LIN {X 0.238,Y -427.107,Z 1023.933,A 0.000,B 0.000,C 90.000,E1 203.823} C_DIS
LIN {X -0.247,Y -422.074,Z 1023.919,A 0.000,B 0.000,C 90.000,E1 201.535} C_DIS
LIN {X 0.239,Y -416.335,Z 1023.903,A 0.000,B 0.000,C 90.000,E1 198.417} C_DIS
LIN {X -0.105,Y -409.408,Z 1023.878,A 0.000,B 0.000,C 90.000,E1 194.008} C_DIS
LIN {X -0.209,Y -406.791,Z 1023.866,A 0.000,B 0.000,C 90.000,E1 191.951} C_DIS
LIN {X -0.089,Y -405.984,Z 1023.860,A 0.000,B 0.000,C 90.000,E1 190.894} C_DIS
LIN {X -0.067,Y -405.858,Z 1023.857,A 0.000,B 0.000,C 90.000,E1 190.197} C_DIS
LIN {X 0.174,Y -406.074,Z 1023.856,A 0.000,B 0.000,C 90.000,E1 189.962} C_DIS
LIN {X 0.195,Y -406.543,Z 1023.852,A 0.000,B 0.000,C 90.000,E1 189.265} C_DIS
LIN {X 0.208,Y -407.205,Z 1023.850,A 0.000,B 0.000,C 90.000,E1 188.916} C_DIS
LIN {X -0.175,Y -408.954,Z 1023.847,A 0.000,B 0.000,C 90.000,E1 188.398} C_DIS
LIN {X -0.116,Y -411.971,Z 1023.843,A 0.000,B 0.000,C 90.000,E1 187.701} C_DIS
LIN {X -0.050,Y -416.031,Z 1023.839,A 0.000,B 0.000,C 90.000,E1 187.004} C_DIS
LIN {X 0.026,Y -419.441,Z 1023.836,A 0.000,B 0.000,C 90.000,E1 186.486} C_DIS
LIN {X -0.081,Y -428.211,Z 1023.830,A 0.000,B 0.000,C 90.000,E1 185.334} C_DIS
LIN {X -0.106,Y -440.088,Z 1023.821,A 0.000,B 0.000,C 90.000,E1 183.841} C_DIS
LIN {X -0.100,Y -449.299,Z 1023.815,A 0.000,B 0.000,C 90.000,E1 182.694} C_DIS
LIN {X -0.039,Y -460.677,Z 1023.807,A 0.000,B 0.000,C 90.000,E1 181.260} C_DIS
LIN {X 0.183,Y -467.926,Z 1023.802,A 0.000,B 0.000,C 90.000,E1 180.286} C_DIS
LIN {X 0.049,Y -474.878,Z 1023.797,A 0.000,B 0.000,C 90.000,E1 179.370} C_DIS
LIN {X 0.054,Y -482.712,Z 1023.791,A 0.000,B 0.000,C 90.000,E1 178.282} C_DIS
LIN {X -0.145,Y -488.160,Z 1023.786,A 0.000,B 0.000,C 90.000,E1 177.535} C_DIS
LIN {X -0.121,Y -494.546,Z 1023.781,A 0.000,B 0.000,C 90.000,E1 176.617} C_DIS
LIN {X -0.011,Y -502.317,Z 1023.775,A 0.000,B 0.000,C 90.000,E1 175.412} C_DIS
LIN {X 0.217,Y -508.156,Z 1023.770,A 0.000,B 0.000,C 90.000,E1 174.489} C_DIS
LIN {X -0.082,Y -515.532,Z 1023.763,A 0.000,B 0.000,C 90.000,E1 173.337} C_DIS
LIN {X -0.238,Y -525.703,Z 1023.753,A 0.000,B 0.000,C 90.000,E1 171.602} C_DIS
LIN {X -0.062,Y -533.859,Z 1023.745,A 0.000,B 0.000,C 90.000,E1 170.151} C_DIS
LIN {X -0.114,Y -541.353,Z 1023.738,A 0.000,B 0.000,C 90.000,E1 168.870} C_DIS
LIN {X -0.051,Y -548.610,Z 1023.731,A 0.000,B 0.000,C 90.000,E1 167.589} C_DIS
LIN {X 0.120,Y -554.019,Z 1023.726,A 0.000,B 0.000,C 90.000,E1 166.589} C_DIS
LIN {X -0.172,Y -561.522,Z 1023.718,A 0.000,B 0.000,C 90.000,E1 165.227} C_DIS
LIN {X -0.068,Y -568.191,Z 1023.711,A 0.000,B 0.000,C 90.000,E1 163.976} C_DIS
LIN {X 0.141,Y -574.462,Z 1023.704,A 0.000,B 0.000,C 90.000,E1 162.725} C_DIS
LIN {X -0.217,Y -578.394,Z 1023.700,A 0.000,B 0.000,C 90.000,E1 161.945} C_DIS
LIN {X 0.119,Y -582.822,Z 1023.694,A 0.000,B 0.000,C 90.000,E1 160.967} C_DIS
LIN {X -0.235,Y -586.875,Z 1023.689,A 0.000,B 0.000,C 90.000,E1 160.061} C_DIS
LIN {X 0.148,Y -591.422,Z 1023.683,A 0.000,B 0.000,C 90.000,E1 158.954} C_DIS
LIN {X -0.174,Y -595.674,Z 1023.677,A 0.000,B 0.000,C 90.000,E1 157.922} C_DIS
LIN {X 0.096,Y -598.641,Z 1023.673,A 0.000,B 0.000,C 90.000,E1 157.102} C_DIS
LIN {X 0.090,Y -602.279,Z 1023.667,A 0.000,B 0.000,C 90.000,E1 156.049} C_DIS
LIN {X -0.170,Y -605.727,Z 1023.661,A 0.000,B 0.000,C 90.000,E1 155.025} C_DIS
LIN {X -0.141,Y -609.702,Z 1023.654,A 0.000,B 0.000,C 90.000,E1 153.717} C_DIS
LIN {X -0.056,Y -613.370,Z 1023.647,A 0.000,B 0.000,C 90.000,E1 152.410} C_DIS
LIN {X -0.166,Y -616.159,Z 1023.641,A 0.000,B 0.000,C 90.000,E1 151.385} C_DIS
LIN {X 0.316,Y -620.763,Z 1023.631,A 0.000,B 0.000,C 90.000,E1 149.537} C_DIS
LIN {X -0.163,Y -626.030,Z 1023.620,A 0.000,B 0.000,C 90.000,E1 147.533} C_DIS
LIN {X 0.163,Y -630.398,Z 1023.610,A 0.000,B 0.000,C 90.000,E1 145.722} C_DIS
LIN {X 0.232,Y -634.076,Z 1023.601,A 0.000,B 0.000,C 90.000,E1 144.196} C_DIS
LIN {X -0.032,Y -636.564,Z 1023.596,A 0.000,B 0.000,C 90.000,E1 143.210} C_DIS
LIN {X 0.009,Y -640.235,Z 1023.587,A 0.000,B 0.000,C 90.000,E1 141.698} C_DIS
LIN {X 0.114,Y -643.267,Z 1023.580,A 0.000,B 0.000,C 90.000,E1 140.436} C_DIS
LIN {X 0.196,Y -646.840,Z 1023.572,A 0.000,B 0.000,C 90.000,E1 138.933} C_DIS
LIN {X 0.175,Y -652.306,Z 1023.560,A 0.000,B 0.000,C 90.000,E1 136.701} C_DIS
LIN {X -0.083,Y -656.221,Z 1023.551,A 0.000,B 0.000,C 90.000,E1 135.243} C_DIS
LIN {X 0.130,Y -664.179,Z 1023.536,A 0.000,B 0.000,C 90.000,E1 132.528} C_DIS
LIN {X 0.143,Y -667.077,Z 1023.531,A 0.000,B 0.000,C 90.000,E1 131.553} C_DIS
LIN {X -0.306,Y -670.039,Z 1023.526,A 0.000,B 0.000,C 90.000,E1 130.620} C_DIS
LIN {X 0.212,Y -672.126,Z 1023.522,A 0.000,B 0.000,C 90.000,E1 129.850} C_DIS
LIN {X -0.089,Y -675.524,Z 1023.515,A 0.000,B 0.000,C 90.000,E1 128.669} C_DIS
LIN {X -0.353,Y -678.146,Z 1023.510,A 0.000,B 0.000,C 90.000,E1 127.729} C_DIS
LIN {X 0.134,Y -682.006,Z 1023.502,A 0.000,B 0.000,C 90.000,E1 126.251} C_DIS
LIN {X 0.150,Y -685.857,Z 1023.494,A 0.000,B 0.000,C 90.000,E1 124.818} C_DIS
LIN {X 0.197,Y -688.889,Z 1023.487,A 0.000,B 0.000,C 90.000,E1 123.627} C_DIS
LIN {X 0.131,Y -692.455,Z 1023.479,A 0.000,B 0.000,C 90.000,E1 122.212} C_DIS
LIN {X 0.249,Y -694.782,Z 1023.474,A 0.000,B 0.000,C 90.000,E1 121.258} C_DIS
LIN {X 0.036,Y -696.837,Z 1023.469,A 0.000,B 0.000,C 90.000,E1 120.335} C_DIS
LIN {X 0.198,Y -698.219,Z 1023.465,A 0.000,B 0.000,C 90.000,E1 119.617} C_DIS
LIN {X 0.032,Y -699.695,Z 1023.459,A 0.000,B 0.000,C 90.000,E1 118.693} C_DIS
LIN {X -0.124,Y -700.907,Z 1023.454,A 0.000,B 0.000,C 90.000,E1 117.769} C_DIS
LIN {X -0.317,Y -701.905,Z 1023.448,A 0.000,B 0.000,C 90.000,E1 116.616} C_DIS
LIN {X 0.141,Y -702.964,Z 1023.441,A 0.000,B 0.000,C 90.000,E1 115.412} C_DIS
LIN {X 0.051,Y -703.422,Z 1023.437,A 0.000,B 0.000,C 90.000,E1 114.719} C_DIS
LIN {X -0.026,Y -703.411,Z 1023.435,A 0.000,B 0.000,C 90.000,E1 114.259} C_DIS
LIN {X -0.033,Y -703.253,Z 1023.434,A 0.000,B 0.000,C 90.000,E1 114.027} C_DIS
LIN {X -0.118,Y -702.452,Z 1023.431,A 0.000,B 0.000,C 90.000,E1 113.567} C_DIS
LIN {X -0.120,Y -701.593,Z 1023.430,A 0.000,B 0.000,C 90.000,E1 113.334} C_DIS
LIN {X 0.149,Y -699.006,Z 1023.427,A 0.000,B 0.000,C 90.000,E1 112.845} C_DIS
LIN {X -0.363,Y -698.118,Z 1023.426,A 0.000,B 0.000,C 90.000,E1 112.770} C_DIS
LIN {X -0.232,Y -696.799,Z 1023.426,A 0.000,B 0.000,C 90.000,E1 112.642} C_DIS
LIN {X 0.181,Y -690.202,Z 1023.424,A 0.000,B 0.000,C 90.000,E1 112.206} C_DIS
LIN {X -0.263,Y -688.193,Z 1023.423,A 0.000,B 0.000,C 90.000,E1 112.153} C_DIS
LIN {X 0.190,Y -685.422,Z 1023.422,A 0.000,B 0.000,C 90.000,E1 112.025} C_DIS
LIN {X 0.156,Y -682.897,Z 1023.422,A 0.000,B 0.000,C 90.000,E1 111.972} C_DIS
LIN {X -0.075,Y -675.659,Z 1023.422,A 0.000,B 0.000,C 90.000,E1 111.897} C_DIS
LIN {X -0.121,Y -614.435,Z 1023.422,A 0.000,B 0.000,C 90.000,E1 111.897} C_DIS
LIN {X 0.287,Y -610.842,Z 1023.421,A 0.000,B 0.000,C 90.000,E1 111.770} C_DIS
LIN {X 0.243,Y -604.194,Z 1023.420,A 0.000,B 0.000,C 90.000,E1 111.535} C_DIS
LIN {X -0.163,Y -598.180,Z 1023.418,A 0.000,B 0.000,C 90.000,E1 111.280} C_DIS
LIN {X 0.284,Y -593.822,Z 1023.417,A 0.000,B 0.000,C 90.000,E1 110.972} C_DIS
LIN {X -0.203,Y -587.457,Z 1023.414,A 0.000,B 0.000,C 90.000,E1 110.556} C_DIS
LIN {X -0.174,Y -576.494,Z 1023.409,A 0.000,B 0.000,C 90.000,E1 109.631} C_DIS
LIN {X 0.317,Y -570.492,Z 1023.407,A 0.000,B 0.000,C 90.000,E1 109.141} C_DIS
LIN {X -0.182,Y -562.239,Z 1023.404,A 0.000,B 0.000,C 90.000,E1 108.725} C_DIS
LIN {X -0.039,Y -555.446,Z 1023.402,A 0.000,B 0.000,C 90.000,E1 108.362} C_DIS
LIN {X 0.238,Y -549.849,Z 1023.400,A 0.000,B 0.000,C 90.000,E1 108.000} C_DIS
LIN {X 0.180,Y -548.206,Z 1023.399,A 0.000,B 0.000,C 90.000,E1 107.819} C_DIS
LIN {X 0.141,Y -548.199,Z 1023.399,A 0.000,B 0.000,C 90.000,E1 107.819} C_DIS
LIN {X -0.010,Y -547.879,Z 1023.398,A 0.000,B 0.000,C 90.000,E1 107.583} C_DIS
LIN {X -0.193,Y -547.944,Z 1023.395,A 0.000,B 0.000,C 90.000,E1 107.040} C_DIS
LIN {X 0.153,Y -548.793,Z 1023.385,A 0.000,B 0.000,C 90.000,E1 105.315} C_DIS
LIN {X 0.104,Y -550.918,Z 1023.367,A 0.000,B 0.000,C 90.000,E1 101.951} C_DIS
LIN {X 0.102,Y -553.715,Z 1023.351,A 0.000,B 0.000,C 90.000,E1 99.151} C_DIS
LIN {X 0.086,Y -555.326,Z 1023.343,A 0.000,B 0.000,C 90.000,E1 97.757} C_DIS
LIN {X 0.080,Y -557.151,Z 1023.334,A 0.000,B 0.000,C 90.000,E1 96.087} C_DIS
LIN {X -0.084,Y -558.195,Z 1023.328,A 0.000,B 0.000,C 90.000,E1 94.992} C_DIS
LIN {X -0.241,Y -559.012,Z 1023.322,A 0.000,B 0.000,C 90.000,E1 93.898} C_DIS
LIN {X 0.217,Y -559.796,Z 1023.314,A 0.000,B 0.000,C 90.000,E1 92.465} C_DIS
LIN {X 0.040,Y -560.284,Z 1023.308,A 0.000,B 0.000,C 90.000,E1 91.375} C_DIS
LIN {X -0.051,Y -560.845,Z 1023.300,A 0.000,B 0.000,C 90.000,E1 90.000} C_DIS
LIN {X -0.035,Y -561.462,Z 1023.291,A 0.000,B 0.000,C 90.000,E1 88.339} C_DIS
LIN {X -0.097,Y -561.895,Z 1023.283,A 0.000,B 0.000,C 90.000,E1 86.963} C_DIS
LIN {X -0.114,Y -562.215,Z 1023.275,A 0.000,B 0.000,C 90.000,E1 85.584} C_DIS
LIN {X 0.023,Y -562.574,Z 1023.266,A 0.000,B 0.000,C 90.000,E1 83.913} C_DIS
LIN {X 0.013,Y -562.852,Z 1023.259,A 0.000,B 0.000,C 90.000,E1 82.534} C_DIS
LIN {X -0.180,Y -563.414,Z 1023.248,A 0.000,B 0.000,C 90.000,E1 80.622} C_DIS
LIN {X 0.236,Y -563.971,Z 1023.239,A 0.000,B 0.000,C 90.000,E1 78.926} C_DIS
LIN {X 0.292,Y -564.935,Z 1023.228,A 0.000,B 0.000,C 90.000,E1 76.992} C_DIS
LIN {X -0.050,Y -566.147,Z 1023.217,A 0.000,B 0.000,C 90.000,E1 75.102} C_DIS
LIN {X 0.276,Y -568.030,Z 1023.204,A 0.000,B 0.000,C 90.000,E1 72.598} C_DIS
LIN {X 0.150,Y -569.219,Z 1023.194,A 0.000,B 0.000,C 90.000,E1 70.967} C_DIS
LIN {X 0.040,Y -570.436,Z 1023.185,A 0.000,B 0.000,C 90.000,E1 69.337} C_DIS
LIN {X -0.176,Y -571.511,Z 1023.176,A 0.000,B 0.000,C 90.000,E1 67.720} C_DIS
LIN {X 0.163,Y -572.445,Z 1023.167,A 0.000,B 0.000,C 90.000,E1 66.049} C_DIS
LIN {X 0.221,Y -573.220,Z 1023.158,A 0.000,B 0.000,C 90.000,E1 64.409} C_DIS
LIN {X 0.035,Y -573.929,Z 1023.149,A 0.000,B 0.000,C 90.000,E1 62.794} C_DIS
LIN {X 0.026,Y -574.487,Z 1023.141,A 0.000,B 0.000,C 90.000,E1 61.435} C_DIS
LIN {X 0.143,Y -575.006,Z 1023.132,A 0.000,B 0.000,C 90.000,E1 59.793} C_DIS
LIN {X -0.070,Y -575.415,Z 1023.125,A 0.000,B 0.000,C 90.000,E1 58.456} C_DIS
LIN {X 0.010,Y -575.978,Z 1023.114,A 0.000,B 0.000,C 90.000,E1 56.548} C_DIS
LIN {X 0.115,Y -576.159,Z 1023.107,A 0.000,B 0.000,C 90.000,E1 55.182} C_DIS
LIN {X -0.077,Y -576.198,Z 1023.101,A 0.000,B 0.000,C 90.000,E1 54.116} C_DIS
LIN {X 0.042,Y -575.983,Z 1023.092,A 0.000,B 0.000,C 90.000,E1 52.477} C_DIS
LIN {X 0.047,Y -575.719,Z 1023.087,A 0.000,B 0.000,C 90.000,E1 51.662} C_DIS
LIN {X -0.017,Y -575.097,Z 1023.080,A 0.000,B 0.000,C 90.000,E1 50.312} C_DIS
LIN {X 0.052,Y -574.456,Z 1023.073,A 0.000,B 0.000,C 90.000,E1 49.218} C_DIS
LIN {X -0.256,Y -573.630,Z 1023.067,A 0.000,B 0.000,C 90.000,E1 48.162} C_DIS
LIN {X 0.100,Y -572.890,Z 1023.063,A 0.000,B 0.000,C 90.000,E1 47.310} C_DIS
LIN {X 0.030,Y -572.034,Z 1023.058,A 0.000,B 0.000,C 90.000,E1 46.500} C_DIS
LIN {X -0.034,Y -571.006,Z 1023.054,A 0.000,B 0.000,C 90.000,E1 45.688} C_DIS
LIN {X 0.278,Y -569.758,Z 1023.049,A 0.000,B 0.000,C 90.000,E1 44.838} C_DIS
LIN {X -0.127,Y -567.825,Z 1023.043,A 0.000,B 0.000,C 90.000,E1 43.785} C_DIS
LIN {X 0.162,Y -566.215,Z 1023.039,A 0.000,B 0.000,C 90.000,E1 42.933} C_DIS
LIN {X 0.017,Y -564.376,Z 1023.034,A 0.000,B 0.000,C 90.000,E1 42.123} C_DIS
LIN {X -0.107,Y -562.280,Z 1023.029,A 0.000,B 0.000,C 90.000,E1 41.310} C_DIS
LIN {X 0.027,Y -560.776,Z 1023.026,A 0.000,B 0.000,C 90.000,E1 40.744} C_DIS
LIN {X -0.130,Y -558.213,Z 1023.022,A 0.000,B 0.000,C 90.000,E1 39.930} C_DIS
LIN {X 0.039,Y -556.400,Z 1023.019,A 0.000,B 0.000,C 90.000,E1 39.358} C_DIS
LIN {X -0.086,Y -552.227,Z 1023.013,A 0.000,B 0.000,C 90.000,E1 38.257} C_DIS
LIN {X 0.109,Y -548.808,Z 1023.008,A 0.000,B 0.000,C 90.000,E1 37.397} C_DIS
LIN {X -0.176,Y -544.975,Z 1023.003,A 0.000,B 0.000,C 90.000,E1 36.583} C_DIS
LIN {X -0.216,Y -540.212,Z 1022.998,A 0.000,B 0.000,C 90.000,E1 35.598} C_DIS
LIN {X 0.279,Y -534.294,Z 1022.991,A 0.000,B 0.000,C 90.000,E1 34.405} C_DIS
LIN {X 0.115,Y -530.323,Z 1022.987,A 0.000,B 0.000,C 90.000,E1 33.706} C_DIS
LIN {X -0.217,Y -526.961,Z 1022.984,A 0.000,B 0.000,C 90.000,E1 33.166} C_DIS
LIN {X 0.110,Y -521.657,Z 1022.979,A 0.000,B 0.000,C 90.000,E1 32.260} C_DIS
LIN {X -0.007,Y -516.913,Z 1022.975,A 0.000,B 0.000,C 90.000,E1 31.544} C_DIS
LIN {X -0.071,Y -510.566,Z 1022.970,A 0.000,B 0.000,C 90.000,E1 30.669} C_DIS
LIN {X -0.091,Y -505.995,Z 1022.967,A 0.000,B 0.000,C 90.000,E1 30.079} C_DIS
LIN {X -0.085,Y -499.845,Z 1022.963,A 0.000,B 0.000,C 90.000,E1 29.333} C_DIS
LIN {X 0.111,Y -490.441,Z 1022.957,A 0.000,B 0.000,C 90.000,E1 28.281} C_DIS
LIN {X -0.058,Y -483.412,Z 1022.953,A 0.000,B 0.000,C 90.000,E1 27.590} C_DIS
LIN {X 0.000,Y -473.405,Z 1022.948,A 0.000,B 0.000,C 90.000,E1 26.616} C_DIS
LIN {X 0.114,Y -467.493,Z 1022.945,A 0.000,B 0.000,C 90.000,E1 26.052} C_DIS
LIN {X -0.104,Y -461.491,Z 1022.942,A 0.000,B 0.000,C 90.000,E1 25.540} C_DIS
LIN {X 0.152,Y -450.872,Z 1022.937,A 0.000,B 0.000,C 90.000,E1 24.591} C_DIS
LIN {X -0.142,Y -428.173,Z 1022.926,A 0.000,B 0.000,C 90.000,E1 22.642} C_DIS
LIN {X 0.106,Y -416.575,Z 1022.919,A 0.000,B 0.000,C 90.000,E1 21.482} C_DIS
LIN {X -0.041,Y -400.990,Z 1022.910,A 0.000,B 0.000,C 90.000,E1 19.812} C_DIS
LIN {X 0.210,Y -398.500,Z 1022.908,A 0.000,B 0.000,C 90.000,E1 19.450} C_DIS
LIN {X -0.085,Y -396.060,Z 1022.906,A 0.000,B 0.000,C 90.000,E1 19.141} C_DIS
LIN {X 0.016,Y -392.977,Z 1022.903,A 0.000,B 0.000,C 90.000,E1 18.598} C_DIS
LIN {X 0.116,Y -391.817,Z 1022.901,A 0.000,B 0.000,C 90.000,E1 18.236} C_DIS
LIN {X 0.165,Y -391.344,Z 1022.899,A 0.000,B 0.000,C 90.000,E1 17.873} C_DIS
LIN {X 0.093,Y -391.026,Z 1022.898,A 0.000,B 0.000,C 90.000,E1 17.528} C_DIS
LIN {X 0.011,Y -391.342,Z 1022.892,A 0.000,B 0.000,C 90.000,E1 16.622} C_DIS
LIN {X 0.084,Y -397.428,Z 1022.863,A 0.000,B 0.000,C 90.000,E1 11.299} C_DIS
LIN {X -0.142,Y -405.123,Z 1022.838,A 0.000,B 0.000,C 90.000,E1 6.777} C_DIS
LIN {X 0.216,Y -410.997,Z 1022.822,A 0.000,B 0.000,C 90.000,E1 3.955} C_DIS
LIN {X -0.196,Y -413.270,Z 1022.816,A 0.000,B 0.000,C 90.000,E1 2.980} C_DIS
LIN {X -0.192,Y -415.154,Z 1022.813,A 0.000,B 0.000,C 90.000,E1 2.293} C_DIS
LIN {X -0.162,Y -417.112,Z 1022.810,A 0.000,B 0.000,C 90.000,E1 1.776} C_DIS
LIN {X -0.155,Y -418.214,Z 1022.809,A 0.000,B 0.000,C 90.000,E1 1.604} C_DIS
LIN {X 0.197,Y -422.306,Z 1022.806,A 0.000,B 0.000,C 90.000,E1 1.031} C_DIS
LIN {X -0.112,Y -424.026,Z 1022.805,A 0.000,B 0.000,C 90.000,E1 0.917} C_DIS
LIN {X -0.053,Y -427.660,Z 1022.804,A 0.000,B 0.000,C 90.000,E1 0.630} C_DIS
LIN {X 0.087,Y -435.228,Z 1022.801,A 0.000,B 0.000,C 90.000,E1 0.172} C_DIS
LIN {X -0.095,Y -451.763,Z 1022.796,A 0.000,B 0.000,C 90.000,E1 359.198} C_DIS
LIN {X -0.214,Y -466.354,Z 1022.791,A 0.000,B 0.000,C 90.000,E1 358.339} C_DIS
LIN {X 0.187,Y -481.031,Z 1022.786,A 0.000,B 0.000,C 90.000,E1 357.421} C_DIS
LIN {X 0.123,Y -490.892,Z 1022.783,A 0.000,B 0.000,C 90.000,E1 356.846} C_DIS
LIN {X -0.081,Y -500.522,Z 1022.779,A 0.000,B 0.000,C 90.000,E1 356.274} C_DIS
LIN {X 0.034,Y -510.075,Z 1022.776,A 0.000,B 0.000,C 90.000,E1 355.641} C_DIS
LIN {X -0.050,Y -519.104,Z 1022.772,A 0.000,B 0.000,C 90.000,E1 355.008} C_DIS
LIN {X -0.014,Y -525.056,Z 1022.770,A 0.000,B 0.000,C 90.000,E1 354.546} C_DIS
LIN {X 0.279,Y -532.268,Z 1022.766,A 0.000,B 0.000,C 90.000,E1 353.913} C_DIS
LIN {X 0.106,Y -537.667,Z 1022.764,A 0.000,B 0.000,C 90.000,E1 353.451} C_DIS
LIN {X 0.226,Y -541.776,Z 1022.762,A 0.000,B 0.000,C 90.000,E1 353.053} C_DIS
LIN {X 0.078,Y -546.974,Z 1022.759,A 0.000,B 0.000,C 90.000,E1 352.534} C_DIS
LIN {X 0.098,Y -553.001,Z 1022.755,A 0.000,B 0.000,C 90.000,E1 351.837} C_DIS
LIN {X -0.194,Y -557.490,Z 1022.752,A 0.000,B 0.000,C 90.000,E1 351.310} C_DIS
LIN {X -0.238,Y -562.419,Z 1022.748,A 0.000,B 0.000,C 90.000,E1 350.622} C_DIS
LIN {X 0.074,Y -566.098,Z 1022.745,A 0.000,B 0.000,C 90.000,E1 350.038} C_DIS
LIN {X -0.197,Y -571.830,Z 1022.739,A 0.000,B 0.000,C 90.000,E1 349.106} C_DIS
LIN {X -0.048,Y -575.659,Z 1022.736,A 0.000,B 0.000,C 90.000,E1 348.409} C_DIS
LIN {X -0.092,Y -580.449,Z 1022.730,A 0.000,B 0.000,C 90.000,E1 347.465} C_DIS
LIN {X 0.265,Y -585.449,Z 1022.724,A 0.000,B 0.000,C 90.000,E1 346.353} C_DIS
LIN {X 0.024,Y -590.708,Z 1022.718,A 0.000,B 0.000,C 90.000,E1 345.172} C_DIS
LIN {X -0.182,Y -594.085,Z 1022.713,A 0.000,B 0.000,C 90.000,E1 344.393} C_DIS
LIN {X 0.206,Y -599.441,Z 1022.706,A 0.000,B 0.000,C 90.000,E1 343.032} C_DIS
LIN {X -0.010,Y -603.448,Z 1022.700,A 0.000,B 0.000,C 90.000,E1 342.000} C_DIS
LIN {X 0.136,Y -608.197,Z 1022.693,A 0.000,B 0.000,C 90.000,E1 340.678} C_DIS
LIN {X 0.041,Y -611.555,Z 1022.687,A 0.000,B 0.000,C 90.000,E1 339.645} C_DIS
LIN {X 0.208,Y -614.682,Z 1022.681,A 0.000,B 0.000,C 90.000,E1 338.592} C_DIS
LIN {X -0.146,Y -617.607,Z 1022.675,A 0.000,B 0.000,C 90.000,E1 337.592} C_DIS
LIN {X 0.115,Y -620.375,Z 1022.670,A 0.000,B 0.000,C 90.000,E1 336.538} C_DIS
LIN {X -0.160,Y -622.912,Z 1022.664,A 0.000,B 0.000,C 90.000,E1 335.537} C_DIS
LIN {X 0.165,Y -625.756,Z 1022.657,A 0.000,B 0.000,C 90.000,E1 334.229} C_DIS
LIN {X -0.304,Y -628.753,Z 1022.648,A 0.000,B 0.000,C 90.000,E1 332.743} C_DIS
LIN {X 0.087,Y -630.482,Z 1022.643,A 0.000,B 0.000,C 90.000,E1 331.691} C_DIS
LIN {X -0.319,Y -632.463,Z 1022.636,A 0.000,B 0.000,C 90.000,E1 330.461} C_DIS
LIN {X 0.125,Y -633.864,Z 1022.630,A 0.000,B 0.000,C 90.000,E1 329.410} C_DIS
LIN {X 0.069,Y -635.328,Z 1022.623,A 0.000,B 0.000,C 90.000,E1 328.152} C_DIS
LIN {X -0.290,Y -637.049,Z 1022.613,A 0.000,B 0.000,C 90.000,E1 326.421} C_DIS
LIN {X 0.009,Y -637.809,Z 1022.608,A 0.000,B 0.000,C 90.000,E1 325.388} C_DIS
LIN {X -0.314,Y -638.516,Z 1022.599,A 0.000,B 0.000,C 90.000,E1 323.909} C_DIS
LIN {X -0.243,Y -638.894,Z 1022.591,A 0.000,B 0.000,C 90.000,E1 322.396} C_DIS
LIN {X -0.170,Y -639.183,Z 1022.583,A 0.000,B 0.000,C 90.000,E1 320.884} C_DIS
LIN {X 0.204,Y -639.766,Z 1022.573,A 0.000,B 0.000,C 90.000,E1 319.094} C_DIS
LIN {X -0.069,Y -640.150,Z 1022.569,A 0.000,B 0.000,C 90.000,E1 318.366} C_DIS
LIN {X -0.159,Y -640.688,Z 1022.559,A 0.000,B 0.000,C 90.000,E1 316.620} C_DIS
LIN {X 0.171,Y -641.423,Z 1022.549,A 0.000,B 0.000,C 90.000,E1 314.838} C_DIS
LIN {X 0.158,Y -642.103,Z 1022.541,A 0.000,B 0.000,C 90.000,E1 313.338} C_DIS
LIN {X -0.161,Y -642.623,Z 1022.535,A 0.000,B 0.000,C 90.000,E1 312.366} C_DIS
LIN {X -0.110,Y -643.169,Z 1022.527,A 0.000,B 0.000,C 90.000,E1 310.862} C_DIS
LIN {X 0.047,Y -643.455,Z 1022.521,A 0.000,B 0.000,C 90.000,E1 309.850} C_DIS
LIN {X 0.115,Y -643.978,Z 1022.512,A 0.000,B 0.000,C 90.000,E1 308.096} C_DIS
LIN {X -0.123,Y -644.128,Z 1022.505,A 0.000,B 0.000,C 90.000,E1 306.870} C_DIS
LIN {X 0.094,Y -644.542,Z 1022.495,A 0.000,B 0.000,C 90.000,E1 305.105} C_DIS
LIN {X -0.054,Y -645.378,Z 1022.481,A 0.000,B 0.000,C 90.000,E1 302.625} C_DIS
LIN {X 0.191,Y -647.649,Z 1022.465,A 0.000,B 0.000,C 90.000,E1 299.617} C_DIS
LIN {X 0.170,Y -650.034,Z 1022.452,A 0.000,B 0.000,C 90.000,E1 297.385} C_DIS
LIN {X 0.073,Y -651.323,Z 1022.445,A 0.000,B 0.000,C 90.000,E1 296.155} C_DIS
LIN {X 0.091,Y -651.987,Z 1022.441,A 0.000,B 0.000,C 90.000,E1 295.412} C_DIS
LIN {X -0.364,Y -652.507,Z 1022.436,A 0.000,B 0.000,C 90.000,E1 294.463} C_DIS
LIN {X -0.158,Y -652.649,Z 1022.433,A 0.000,B 0.000,C 90.000,E1 293.951} C_DIS
LIN {X -0.015,Y -652.688,Z 1022.428,A 0.000,B 0.000,C 90.000,E1 292.950} C_DIS
LIN {X -0.120,Y -652.493,Z 1022.422,A 0.000,B 0.000,C 90.000,E1 291.972} C_DIS
LIN {X -0.024,Y -652.333,Z 1022.421,A 0.000,B 0.000,C 90.000,E1 291.716} C_DIS
LIN {X -0.076,Y -651.672,Z 1022.418,A 0.000,B 0.000,C 90.000,E1 291.227} C_DIS
LIN {X 0.015,Y -651.139,Z 1022.417,A 0.000,B 0.000,C 90.000,E1 290.972} C_DIS
LIN {X -0.130,Y -650.454,Z 1022.415,A 0.000,B 0.000,C 90.000,E1 290.737} C_DIS
LIN {X -0.046,Y -649.538,Z 1022.414,A 0.000,B 0.000,C 90.000,E1 290.482} C_DIS
LIN {X -0.153,Y -647.125,Z 1022.412,A 0.000,B 0.000,C 90.000,E1 290.120} C_DIS
LIN {X -0.083,Y -645.281,Z 1022.410,A 0.000,B 0.000,C 90.000,E1 289.866} C_DIS
LIN {X -0.269,Y -643.850,Z 1022.410,A 0.000,B 0.000,C 90.000,E1 289.758} C_DIS
LIN {X 0.289,Y -637.928,Z 1022.407,A 0.000,B 0.000,C 90.000,E1 289.268} C_DIS
LIN {X -0.125,Y -629.077,Z 1022.405,A 0.000,B 0.000,C 90.000,E1 288.852} C_DIS
LIN {X -0.114,Y -620.323,Z 1022.403,A 0.000,B 0.000,C 90.000,E1 288.489} C_DIS
LIN {X -0.078,Y -614.966,Z 1022.402,A 0.000,B 0.000,C 90.000,E1 288.290} C_DIS
LIN {X -0.120,Y -614.892,Z 1022.402,A 0.000,B 0.000,C 90.000,E1 288.290} C_DIS
LIN {X -0.048,Y -613.830,Z 1022.401,A 0.000,B 0.000,C 90.000,E1 288.181} C_DIS
LIN {X -0.091,Y -613.796,Z 1022.401,A 0.000,B 0.000,C 90.000,E1 288.181} C_DIS
LIN {X 0.188,Y -614.746,Z 1022.400,A 0.000,B 0.000,C 90.000,E1 287.946} C_DIS
LIN {X -0.135,Y -620.302,Z 1022.396,A 0.000,B 0.000,C 90.000,E1 287.330} C_DIS
LIN {X -0.011,Y -625.332,Z 1022.393,A 0.000,B 0.000,C 90.000,E1 286.677} C_DIS
LIN {X -0.223,Y -627.049,Z 1022.391,A 0.000,B 0.000,C 90.000,E1 286.441} C_DIS
LIN {X 0.148,Y -630.271,Z 1022.388,A 0.000,B 0.000,C 90.000,E1 285.898} C_DIS
LIN {X -0.247,Y -633.695,Z 1022.385,A 0.000,B 0.000,C 90.000,E1 285.300} C_DIS
LIN {X -0.009,Y -636.406,Z 1022.381,A 0.000,B 0.000,C 90.000,E1 284.647} C_DIS
LIN {X -0.186,Y -637.428,Z 1022.380,A 0.000,B 0.000,C 90.000,E1 284.411} C_DIS
LIN {X 0.088,Y -638.952,Z 1022.377,A 0.000,B 0.000,C 90.000,E1 283.883} C_DIS
LIN {X 0.214,Y -640.736,Z 1022.373,A 0.000,B 0.000,C 90.000,E1 283.119} C_DIS
LIN {X -0.108,Y -641.350,Z 1022.370,A 0.000,B 0.000,C 90.000,E1 282.647} C_DIS
LIN {X 0.200,Y -641.652,Z 1022.367,A 0.000,B 0.000,C 90.000,E1 282.119} C_DIS
LIN {X -0.249,Y -641.696,Z 1022.365,A 0.000,B 0.000,C 90.000,E1 281.658} C_DIS
LIN {X 0.223,Y -641.623,Z 1022.363,A 0.000,B 0.000,C 90.000,E1 281.366} C_DIS
LIN {X -0.095,Y -641.166,Z 1022.361,A 0.000,B 0.000,C 90.000,E1 280.894} C_DIS
LIN {X 0.209,Y -640.299,Z 1022.358,A 0.000,B 0.000,C 90.000,E1 280.366} C_DIS
LIN {X -0.069,Y -639.739,Z 1022.356,A 0.000,B 0.000,C 90.000,E1 280.141} C_DIS
LIN {X 0.225,Y -638.276,Z 1022.354,A 0.000,B 0.000,C 90.000,E1 279.613} C_DIS
LIN {X -0.226,Y -636.288,Z 1022.351,A 0.000,B 0.000,C 90.000,E1 279.151} C_DIS
LIN {X -0.102,Y -633.257,Z 1022.347,A 0.000,B 0.000,C 90.000,E1 278.511} C_DIS
LIN {X 0.045,Y -630.213,Z 1022.344,A 0.000,B 0.000,C 90.000,E1 277.992} C_DIS
LIN {X -0.304,Y -627.169,Z 1022.342,A 0.000,B 0.000,C 90.000,E1 277.644} C_DIS
LIN {X -0.046,Y -623.879,Z 1022.340,A 0.000,B 0.000,C 90.000,E1 277.239} C_DIS
LIN {X -0.133,Y -620.612,Z 1022.338,A 0.000,B 0.000,C 90.000,E1 276.891} C_DIS
LIN {X 0.128,Y -613.844,Z 1022.335,A 0.000,B 0.000,C 90.000,E1 276.258} C_DIS
LIN {X -0.174,Y -606.418,Z 1022.332,A 0.000,B 0.000,C 90.000,E1 275.739} C_DIS
LIN {X -0.120,Y -600.055,Z 1022.330,A 0.000,B 0.000,C 90.000,E1 275.334} C_DIS
LIN {X 0.232,Y -596.360,Z 1022.329,A 0.000,B 0.000,C 90.000,E1 275.106} C_DIS
LIN {X -0.273,Y -593.117,Z 1022.328,A 0.000,B 0.000,C 90.000,E1 274.992} C_DIS
LIN {X 0.114,Y -585.759,Z 1022.326,A 0.000,B 0.000,C 90.000,E1 274.645} C_DIS
LIN {X -0.007,Y -579.116,Z 1022.325,A 0.000,B 0.000,C 90.000,E1 274.473} C_DIS
LIN {X -0.156,Y -573.305,Z 1022.324,A 0.000,B 0.000,C 90.000,E1 274.359} C_DIS
LIN {X -0.062,Y -566.759,Z 1022.324,A 0.000,B 0.000,C 90.000,E1 274.245} C_DIS
LIN {X -0.240,Y -564.290,Z 1022.323,A 0.000,B 0.000,C 90.000,E1 274.245} C_DIS
LIN {X -0.283,Y -561.291,Z 1022.323,A 0.000,B 0.000,C 90.000,E1 274.245} C_DIS
LIN {X 0.226,Y -543.993,Z 1022.323,A 0.000,B 0.000,C 90.000,E1 274.188} C_DIS
LIN {X 0.205,Y -543.044,Z 1022.322,A 0.000,B 0.000,C 90.000,E1 273.898} C_DIS
LIN {X -0.149,Y -542.751,Z 1022.321,A 0.000,B 0.000,C 90.000,E1 273.784} C_DIS
LIN {X -0.022,Y -541.589,Z 1022.315,A 0.000,B 0.000,C 90.000,E1 272.636} C_DIS
LIN {X 0.155,Y -540.547,Z 1022.304,A 0.000,B 0.000,C 90.000,E1 270.630} C_DIS
LIN {X 0.240,Y -539.881,Z 1022.297,A 0.000,B 0.000,C 90.000,E1 269.484} C_DIS
LIN {X -0.229,Y -539.085,Z 1022.291,A 0.000,B 0.000,C 90.000,E1 268.396} C_DIS
LIN {X -0.108,Y -537.766,Z 1022.281,A 0.000,B 0.000,C 90.000,E1 266.674} C_DIS
LIN {X -0.011,Y -536.281,Z 1022.270,A 0.000,B 0.000,C 90.000,E1 264.666} C_DIS
LIN {X 0.108,Y -535.164,Z 1022.262,A 0.000,B 0.000,C 90.000,E1 263.223} C_DIS
LIN {X 0.185,Y -534.473,Z 1022.258,A 0.000,B 0.000,C 90.000,E1 262.356} C_DIS
LIN {X -0.226,Y -533.329,Z 1022.251,A 0.000,B 0.000,C 90.000,E1 261.254} C_DIS
LIN {X -0.126,Y -532.008,Z 1022.245,A 0.000,B 0.000,C 90.000,E1 260.095} C_DIS
LIN {X 0.200,Y -529.460,Z 1022.232,A 0.000,B 0.000,C 90.000,E1 257.757} C_DIS
LIN {X -0.005,Y -527.599,Z 1022.223,A 0.000,B 0.000,C 90.000,E1 256.047} C_DIS
LIN {X 0.220,Y -526.292,Z 1022.216,A 0.000,B 0.000,C 90.000,E1 254.866} C_DIS
LIN {X 0.077,Y -524.091,Z 1022.205,A 0.000,B 0.000,C 90.000,E1 252.851} C_DIS
LIN {X 0.032,Y -522.555,Z 1022.197,A 0.000,B 0.000,C 90.000,E1 251.402} C_DIS
LIN {X 0.106,Y -520.323,Z 1022.187,A 0.000,B 0.000,C 90.000,E1 249.645} C_DIS
LIN {X -0.178,Y -517.985,Z 1022.177,A 0.000,B 0.000,C 90.000,E1 247.922} C_DIS
LIN {X -0.312,Y -515.645,Z 1022.167,A 0.000,B 0.000,C 90.000,E1 246.177} C_DIS
LIN {X -0.062,Y -513.916,Z 1022.161,A 0.000,B 0.000,C 90.000,E1 244.973} C_DIS
LIN {X 0.165,Y -512.160,Z 1022.154,A 0.000,B 0.000,C 90.000,E1 243.768} C_DIS
LIN {X -0.097,Y -510.283,Z 1022.148,A 0.000,B 0.000,C 90.000,E1 242.615} C_DIS
LIN {X -0.181,Y -507.264,Z 1022.138,A 0.000,B 0.000,C 90.000,E1 240.845} C_DIS
LIN {X 0.045,Y -504.639,Z 1022.130,A 0.000,B 0.000,C 90.000,E1 239.331} C_DIS
LIN {X 0.166,Y -502.381,Z 1022.123,A 0.000,B 0.000,C 90.000,E1 238.122} C_DIS
LIN {X -0.169,Y -500.079,Z 1022.116,A 0.000,B 0.000,C 90.000,E1 236.962} C_DIS
LIN {X 0.155,Y -497.489,Z 1022.110,A 0.000,B 0.000,C 90.000,E1 235.722} C_DIS
LIN {X 0.029,Y -494.756,Z 1022.103,A 0.000,B 0.000,C 90.000,E1 234.529} C_DIS
LIN {X 0.107,Y -491.182,Z 1022.095,A 0.000,B 0.000,C 90.000,E1 233.004} C_DIS
LIN {X 0.006,Y -487.528,Z 1022.086,A 0.000,B 0.000,C 90.000,E1 231.492} C_DIS
LIN {X -0.283,Y -482.585,Z 1022.074,A 0.000,B 0.000,C 90.000,E1 229.380} C_DIS
LIN {X 0.186,Y -478.445,Z 1022.064,A 0.000,B 0.000,C 90.000,E1 227.472} C_DIS
LIN {X -0.143,Y -474.486,Z 1022.054,A 0.000,B 0.000,C 90.000,E1 225.648} C_DIS
LIN {X 0.256,Y -471.990,Z 1022.047,A 0.000,B 0.000,C 90.000,E1 224.352} C_DIS
LIN {X -0.141,Y -467.438,Z 1022.034,A 0.000,B 0.000,C 90.000,E1 222.204} C_DIS
LIN {X -0.030,Y -463.579,Z 1022.024,A 0.000,B 0.000,C 90.000,E1 220.297} C_DIS
LIN {X -0.089,Y -460.832,Z 1022.017,A 0.000,B 0.000,C 90.000,E1 219.036} C_DIS
LIN {X -0.093,Y -457.192,Z 1022.008,A 0.000,B 0.000,C 90.000,E1 217.443} C_DIS
LIN {X 0.010,Y -452.258,Z 1021.996,A 0.000,B 0.000,C 90.000,E1 215.185} C_DIS
LIN {X 0.022,Y -448.070,Z 1021.985,A 0.000,B 0.000,C 90.000,E1 213.245} C_DIS
LIN {X 0.070,Y -443.820,Z 1021.974,A 0.000,B 0.000,C 90.000,E1 211.288} C_DIS
LIN {X -0.084,Y -441.018,Z 1021.967,A 0.000,B 0.000,C 90.000,E1 210.001} C_DIS
LIN {X -0.089,Y -437.298,Z 1021.958,A 0.000,B 0.000,C 90.000,E1 208.359} C_DIS
LIN {X 0.027,Y -432.773,Z 1021.947,A 0.000,B 0.000,C 90.000,E1 206.360} C_DIS
LIN {X 0.037,Y -427.519,Z 1021.934,A 0.000,B 0.000,C 90.000,E1 204.027} C_DIS
LIN {X -0.057,Y -423.111,Z 1021.922,A 0.000,B 0.000,C 90.000,E1 202.025} C_DIS
LIN {X 0.069,Y -417.200,Z 1021.905,A 0.000,B 0.000,C 90.000,E1 198.960} C_DIS
LIN {X -0.004,Y -411.431,Z 1021.886,A 0.000,B 0.000,C 90.000,E1 195.552} C_DIS
LIN {X 0.036,Y -408.501,Z 1021.875,A 0.000,B 0.000,C 90.000,E1 193.480} C_DIS
LIN {X -0.103,Y -406.324,Z 1021.865,A 0.000,B 0.000,C 90.000,E1 191.771} C_DIS
LIN {X 0.008,Y -405.348,Z 1021.860,A 0.000,B 0.000,C 90.000,E1 190.715} C_DIS
LIN {X 0.024,Y -405.135,Z 1021.856,A 0.000,B 0.000,C 90.000,E1 190.018} C_DIS
LIN {X 0.038,Y -405.583,Z 1021.852,A 0.000,B 0.000,C 90.000,E1 189.321} C_DIS
LIN {X 0.041,Y -406.374,Z 1021.849,A 0.000,B 0.000,C 90.000,E1 188.803} C_DIS
LIN {X 0.077,Y -406.760,Z 1021.848,A 0.000,B 0.000,C 90.000,E1 188.624} C_DIS
LIN {X 0.093,Y -408.617,Z 1021.845,A 0.000,B 0.000,C 90.000,E1 188.049} C_DIS
LIN {X 0.146,Y -410.722,Z 1021.842,A 0.000,B 0.000,C 90.000,E1 187.530} C_DIS
LIN {X 0.146,Y -415.197,Z 1021.838,A 0.000,B 0.000,C 90.000,E1 186.720} C_DIS
LIN {X 0.182,Y -423.338,Z 1021.831,A 0.000,B 0.000,C 90.000,E1 185.568} C_DIS
LIN {X -0.060,Y -436.424,Z 1021.822,A 0.000,B 0.000,C 90.000,E1 183.955} C_DIS
LIN {X 0.025,Y -444.284,Z 1021.817,A 0.000,B 0.000,C 90.000,E1 182.980} C_DIS
LIN {X 0.188,Y -455.777,Z 1021.809,A 0.000,B 0.000,C 90.000,E1 181.547} C_DIS
LIN {X -0.165,Y -463.385,Z 1021.803,A 0.000,B 0.000,C 90.000,E1 180.630} C_DIS
LIN {X 0.200,Y -471.750,Z 1021.797,A 0.000,B 0.000,C 90.000,E1 179.484} C_DIS
LIN {X -0.066,Y -477.482,Z 1021.793,A 0.000,B 0.000,C 90.000,E1 178.740} C_DIS
LIN {X 0.169,Y -483.154,Z 1021.789,A 0.000,B 0.000,C 90.000,E1 177.936} C_DIS
LIN {X -0.044,Y -488.650,Z 1021.784,A 0.000,B 0.000,C 90.000,E1 177.192} C_DIS
LIN {X 0.015,Y -495.018,Z 1021.779,A 0.000,B 0.000,C 90.000,E1 176.274} C_DIS
LIN {X -0.201,Y -501.958,Z 1021.773,A 0.000,B 0.000,C 90.000,E1 175.241} C_DIS
LIN {X 0.214,Y -508.758,Z 1021.768,A 0.000,B 0.000,C 90.000,E1 174.147} C_DIS
LIN {X -0.083,Y -516.156,Z 1021.761,A 0.000,B 0.000,C 90.000,E1 172.996} C_DIS
LIN {X 0.012,Y -525.523,Z 1021.752,A 0.000,B 0.000,C 90.000,E1 171.376} C_DIS
LIN {X 0.057,Y -533.780,Z 1021.744,A 0.000,B 0.000,C 90.000,E1 169.926} C_DIS
LIN {X 0.032,Y -539.695,Z 1021.739,A 0.000,B 0.000,C 90.000,E1 168.926} C_DIS
LIN {X -0.183,Y -546.209,Z 1021.732,A 0.000,B 0.000,C 90.000,E1 167.813} C_DIS
LIN {X -0.161,Y -551.724,Z 1021.727,A 0.000,B 0.000,C 90.000,E1 166.825} C_DIS
LIN {X 0.045,Y -559.308,Z 1021.719,A 0.000,B 0.000,C 90.000,E1 165.408} C_DIS
LIN {X -0.003,Y -566.825,Z 1021.711,A 0.000,B 0.000,C 90.000,E1 164.031} C_DIS
LIN {X 0.189,Y -573.142,Z 1021.704,A 0.000,B 0.000,C 90.000,E1 162.779} C_DIS
LIN {X 0.280,Y -577.766,Z 1021.699,A 0.000,B 0.000,C 90.000,E1 161.819} C_DIS
LIN {X 0.270,Y -583.460,Z 1021.692,A 0.000,B 0.000,C 90.000,E1 160.604} C_DIS
LIN {X 0.275,Y -589.203,Z 1021.685,A 0.000,B 0.000,C 90.000,E1 159.263} C_DIS
LIN {X -0.073,Y -593.595,Z 1021.679,A 0.000,B 0.000,C 90.000,E1 158.230} C_DIS
LIN {X 0.172,Y -596.711,Z 1021.675,A 0.000,B 0.000,C 90.000,E1 157.411} C_DIS
LIN {X 0.143,Y -600.463,Z 1021.669,A 0.000,B 0.000,C 90.000,E1 156.357} C_DIS
LIN {X 0.157,Y -604.015,Z 1021.663,A 0.000,B 0.000,C 90.000,E1 155.305} C_DIS
LIN {X -0.133,Y -608.108,Z 1021.656,A 0.000,B 0.000,C 90.000,E1 154.024} C_DIS
LIN {X -0.350,Y -611.890,Z 1021.648,A 0.000,B 0.000,C 90.000,E1 152.743} C_DIS
LIN {X -0.194,Y -614.754,Z 1021.643,A 0.000,B 0.000,C 90.000,E1 151.691} C_DIS
LIN {X -0.043,Y -619.401,Z 1021.633,A 0.000,B 0.000,C 90.000,E1 149.871} C_DIS
LIN {X -0.021,Y -624.001,Z 1021.623,A 0.000,B 0.000,C 90.000,E1 148.074} C_DIS
LIN {X -0.238,Y -625.948,Z 1021.618,A 0.000,B 0.000,C 90.000,E1 147.327} C_DIS
LIN {X -0.266,Y -629.768,Z 1021.610,A 0.000,B 0.000,C 90.000,E1 145.801} C_DIS
LIN {X -0.216,Y -633.482,Z 1021.602,A 0.000,B 0.000,C 90.000,E1 144.276} C_DIS
LIN {X -0.112,Y -636.014,Z 1021.596,A 0.000,B 0.000,C 90.000,E1 143.256} C_DIS
LIN {X -0.072,Y -639.706,Z 1021.587,A 0.000,B 0.000,C 90.000,E1 141.743} C_DIS
LIN {X 0.033,Y -642.776,Z 1021.581,A 0.000,B 0.000,C 90.000,E1 140.481} C_DIS
LIN {X 0.189,Y -645.758,Z 1021.574,A 0.000,B 0.000,C 90.000,E1 139.218} C_DIS
LIN {X -0.034,Y -648.167,Z 1021.568,A 0.000,B 0.000,C 90.000,E1 138.243} C_DIS
LIN {X 0.002,Y -653.131,Z 1021.557,A 0.000,B 0.000,C 90.000,E1 136.257} C_DIS
LIN {X 0.273,Y -656.467,Z 1021.550,A 0.000,B 0.000,C 90.000,E1 135.000} C_DIS
LIN {X 0.040,Y -663.029,Z 1021.538,A 0.000,B 0.000,C 90.000,E1 132.813} C_DIS
LIN {X 0.030,Y -666.047,Z 1021.532,A 0.000,B 0.000,C 90.000,E1 131.838} C_DIS
LIN {X 0.070,Y -669.711,Z 1021.526,A 0.000,B 0.000,C 90.000,E1 130.620} C_DIS
LIN {X 0.155,Y -671.844,Z 1021.522,A 0.000,B 0.000,C 90.000,E1 129.886} C_DIS
LIN {X 0.282,Y -675.249,Z 1021.515,A 0.000,B 0.000,C 90.000,E1 128.669} C_DIS
LIN {X 0.015,Y -677.911,Z 1021.510,A 0.000,B 0.000,C 90.000,E1 127.729} C_DIS
LIN {X -0.049,Y -681.791,Z 1021.502,A 0.000,B 0.000,C 90.000,E1 126.297} C_DIS
LIN {X -0.049,Y -685.649,Z 1021.494,A 0.000,B 0.000,C 90.000,E1 124.865} C_DIS
LIN {X -0.025,Y -688.117,Z 1021.488,A 0.000,B 0.000,C 90.000,E1 123.913} C_DIS
LIN {X -0.104,Y -691.693,Z 1021.481,A 0.000,B 0.000,C 90.000,E1 122.498} C_DIS
LIN {X -0.345,Y -694.624,Z 1021.474,A 0.000,B 0.000,C 90.000,E1 121.337} C_DIS
LIN {X -0.206,Y -696.701,Z 1021.469,A 0.000,B 0.000,C 90.000,E1 120.384} C_DIS
LIN {X -0.050,Y -698.112,Z 1021.465,A 0.000,B 0.000,C 90.000,E1 119.667} C_DIS
LIN {X -0.223,Y -699.600,Z 1021.460,A 0.000,B 0.000,C 90.000,E1 118.743} C_DIS
LIN {X -0.036,Y -700.570,Z 1021.456,A 0.000,B 0.000,C 90.000,E1 118.025} C_DIS
LIN {X -0.163,Y -701.240,Z 1021.452,A 0.000,B 0.000,C 90.000,E1 117.334} C_DIS
LIN {X -0.138,Y -702.884,Z 1021.441,A 0.000,B 0.000,C 90.000,E1 115.463} C_DIS
LIN {X -0.232,Y -703.357,Z 1021.438,A 0.000,B 0.000,C 90.000,E1 114.771} C_DIS
LIN {X 0.329,Y -703.353,Z 1021.435,A 0.000,B 0.000,C 90.000,E1 114.259} C_DIS
LIN {X -0.321,Y -703.240,Z 1021.434,A 0.000,B 0.000,C 90.000,E1 114.079} C_DIS
LIN {X -0.044,Y -702.471,Z 1021.431,A 0.000,B 0.000,C 90.000,E1 113.590} C_DIS
LIN {X 0.233,Y -701.719,Z 1021.430,A 0.000,B 0.000,C 90.000,E1 113.334} C_DIS
LIN {X -0.142,Y -699.141,Z 1021.427,A 0.000,B 0.000,C 90.000,E1 112.898} C_DIS
LIN {X -0.010,Y -698.335,Z 1021.427,A 0.000,B 0.000,C 90.000,E1 112.770} C_DIS
LIN {X 0.121,Y -697.137,Z 1021.426,A 0.000,B 0.000,C 90.000,E1 112.642} C_DIS
LIN {X -0.043,Y -692.014,Z 1021.424,A 0.000,B 0.000,C 90.000,E1 112.333} C_DIS
LIN {X 0.410,Y -690.519,Z 1021.424,A 0.000,B 0.000,C 90.000,E1 112.206} C_DIS
LIN {X -0.029,Y -688.737,Z 1021.423,A 0.000,B 0.000,C 90.000,E1 112.153} C_DIS
LIN {X -0.251,Y -684.078,Z 1021.422,A 0.000,B 0.000,C 90.000,E1 112.025} C_DIS
LIN {X -0.009,Y -676.347,Z 1021.422,A 0.000,B 0.000,C 90.000,E1 111.897} C_DIS
LIN {X -0.152,Y -674.771,Z 1021.422,A 0.000,B 0.000,C 90.000,E1 111.897} C_DIS
LIN {X -0.189,Y -614.811,Z 1021.422,A 0.000,B 0.000,C 90.000,E1 111.897} C_DIS
LIN {X -0.094,Y -610.266,Z 1021.421,A 0.000,B 0.000,C 90.000,E1 111.770} C_DIS
LIN {X -0.151,Y -604.958,Z 1021.420,A 0.000,B 0.000,C 90.000,E1 111.589} C_DIS
LIN {X -0.053,Y -598.674,Z 1021.418,A 0.000,B 0.000,C 90.000,E1 111.280} C_DIS
LIN {X -0.025,Y -592.850,Z 1021.416,A 0.000,B 0.000,C 90.000,E1 110.918} C_DIS
LIN {X 0.192,Y -587.234,Z 1021.414,A 0.000,B 0.000,C 90.000,E1 110.482} C_DIS
LIN {X 0.060,Y -577.850,Z 1021.410,A 0.000,B 0.000,C 90.000,E1 109.704} C_DIS
LIN {X 0.146,Y -570.398,Z 1021.406,A 0.000,B 0.000,C 90.000,E1 109.141} C_DIS
LIN {X 0.129,Y -561.953,Z 1021.404,A 0.000,B 0.000,C 90.000,E1 108.671} C_DIS
LIN {X -0.222,Y -555.240,Z 1021.402,A 0.000,B 0.000,C 90.000,E1 108.362} C_DIS
LIN {X 0.053,Y -549.652,Z 1021.400,A 0.000,B 0.000,C 90.000,E1 108.000} C_DIS
LIN {X 0.199,Y -548.293,Z 1021.399,A 0.000,B 0.000,C 90.000,E1 107.819} C_DIS
LIN {X 0.157,Y -548.279,Z 1021.399,A 0.000,B 0.000,C 90.000,E1 107.819} C_DIS
LIN {X 0.196,Y -547.932,Z 1021.397,A 0.000,B 0.000,C 90.000,E1 107.402} C_DIS
LIN {X -0.302,Y -548.184,Z 1021.392,A 0.000,B 0.000,C 90.000,E1 106.622} C_DIS
LIN {X -0.050,Y -548.896,Z 1021.384,A 0.000,B 0.000,C 90.000,E1 105.190} C_DIS
LIN {X 0.001,Y -551.303,Z 1021.364,A 0.000,B 0.000,C 90.000,E1 101.535} C_DIS
LIN {X -0.125,Y -553.912,Z 1021.350,A 0.000,B 0.000,C 90.000,E1 99.029} C_DIS
LIN {X 0.157,Y -554.868,Z 1021.345,A 0.000,B 0.000,C 90.000,E1 98.163} C_DIS
LIN {X 0.267,Y -557.028,Z 1021.335,A 0.000,B 0.000,C 90.000,E1 96.201} C_DIS
LIN {X 0.174,Y -558.317,Z 1021.327,A 0.000,B 0.000,C 90.000,E1 94.821} C_DIS
LIN {X 0.021,Y -559.094,Z 1021.321,A 0.000,B 0.000,C 90.000,E1 93.726} C_DIS
LIN {X -0.164,Y -559.752,Z 1021.315,A 0.000,B 0.000,C 90.000,E1 92.636} C_DIS
LIN {X -0.159,Y -560.461,Z 1021.305,A 0.000,B 0.000,C 90.000,E1 90.974} C_DIS
LIN {X -0.245,Y -560.991,Z 1021.298,A 0.000,B 0.000,C 90.000,E1 89.599} C_DIS
LIN {X 0.235,Y -561.551,Z 1021.290,A 0.000,B 0.000,C 90.000,E1 88.167} C_DIS
LIN {X -0.016,Y -561.794,Z 1021.285,A 0.000,B 0.000,C 90.000,E1 87.364} C_DIS
LIN {X 0.063,Y -562.197,Z 1021.276,A 0.000,B 0.000,C 90.000,E1 85.698} C_DIS
LIN {X -0.271,Y -562.572,Z 1021.265,A 0.000,B 0.000,C 90.000,E1 83.799} C_DIS
LIN {X -0.211,Y -562.858,Z 1021.258,A 0.000,B 0.000,C 90.000,E1 82.413} C_DIS
LIN {X 0.007,Y -563.353,Z 1021.249,A 0.000,B 0.000,C 90.000,E1 80.735} C_DIS
LIN {X -0.073,Y -563.996,Z 1021.238,A 0.000,B 0.000,C 90.000,E1 78.814} C_DIS
LIN {X -0.025,Y -564.988,Z 1021.227,A 0.000,B 0.000,C 90.000,E1 76.881} C_DIS
LIN {X 0.172,Y -566.183,Z 1021.216,A 0.000,B 0.000,C 90.000,E1 74.936} C_DIS
LIN {X 0.157,Y -567.660,Z 1021.206,A 0.000,B 0.000,C 90.000,E1 73.015} C_DIS
LIN {X -0.109,Y -568.484,Z 1021.200,A 0.000,B 0.000,C 90.000,E1 71.945} C_DIS
LIN {X -0.045,Y -569.671,Z 1021.191,A 0.000,B 0.000,C 90.000,E1 70.296} C_DIS
LIN {X -0.115,Y -570.457,Z 1021.185,A 0.000,B 0.000,C 90.000,E1 69.209} C_DIS
LIN {X -0.153,Y -571.370,Z 1021.177,A 0.000,B 0.000,C 90.000,E1 67.847} C_DIS
LIN {X 0.180,Y -572.328,Z 1021.168,A 0.000,B 0.000,C 90.000,E1 66.177} C_DIS
LIN {X 0.074,Y -573.228,Z 1021.157,A 0.000,B 0.000,C 90.000,E1 64.280} C_DIS
LIN {X -0.112,Y -573.899,Z 1021.148,A 0.000,B 0.000,C 90.000,E1 62.666} C_DIS
LIN {X -0.123,Y -574.423,Z 1021.141,A 0.000,B 0.000,C 90.000,E1 61.307} C_DIS
LIN {X 0.150,Y -574.869,Z 1021.133,A 0.000,B 0.000,C 90.000,E1 59.921} C_DIS
LIN {X -0.062,Y -575.271,Z 1021.125,A 0.000,B 0.000,C 90.000,E1 58.584} C_DIS
LIN {X -0.299,Y -575.789,Z 1021.115,A 0.000,B 0.000,C 90.000,E1 56.707} C_DIS
LIN {X -0.027,Y -575.967,Z 1021.109,A 0.000,B 0.000,C 90.000,E1 55.595} C_DIS
LIN {X -0.068,Y -576.056,Z 1021.101,A 0.000,B 0.000,C 90.000,E1 54.242} C_DIS
LIN {X 0.054,Y -575.832,Z 1021.092,A 0.000,B 0.000,C 90.000,E1 52.603} C_DIS
LIN {X -0.296,Y -575.576,Z 1021.088,A 0.000,B 0.000,C 90.000,E1 51.823} C_DIS
LIN {X -0.144,Y -575.091,Z 1021.082,A 0.000,B 0.000,C 90.000,E1 50.723} C_DIS
LIN {X -0.005,Y -574.507,Z 1021.076,A 0.000,B 0.000,C 90.000,E1 49.622} C_DIS
LIN {X 0.199,Y -573.515,Z 1021.068,A 0.000,B 0.000,C 90.000,E1 48.243} C_DIS
LIN {X 0.257,Y -572.492,Z 1021.062,A 0.000,B 0.000,C 90.000,E1 47.148} C_DIS
LIN {X -0.211,Y -571.571,Z 1021.058,A 0.000,B 0.000,C 90.000,E1 46.377} C_DIS
LIN {X -0.292,Y -570.491,Z 1021.053,A 0.000,B 0.000,C 90.000,E1 45.567} C_DIS
LIN {X 0.018,Y -569.193,Z 1021.048,A 0.000,B 0.000,C 90.000,E1 44.717} C_DIS
LIN {X 0.008,Y -567.217,Z 1021.042,A 0.000,B 0.000,C 90.000,E1 43.623} C_DIS
LIN {X 0.290,Y -565.527,Z 1021.038,A 0.000,B 0.000,C 90.000,E1 42.771} C_DIS
LIN {X -0.242,Y -563.578,Z 1021.033,A 0.000,B 0.000,C 90.000,E1 42.000} C_DIS
LIN {X 0.001,Y -561.412,Z 1021.029,A 0.000,B 0.000,C 90.000,E1 41.148} C_DIS
LIN {X -0.237,Y -559.810,Z 1021.026,A 0.000,B 0.000,C 90.000,E1 40.620} C_DIS
LIN {X 0.302,Y -558.102,Z 1021.023,A 0.000,B 0.000,C 90.000,E1 40.011} C_DIS
LIN {X 0.120,Y -555.276,Z 1021.018,A 0.000,B 0.000,C 90.000,E1 39.197} C_DIS
LIN {X -0.025,Y -550.994,Z 1021.012,A 0.000,B 0.000,C 90.000,E1 38.096} C_DIS
LIN {X -0.041,Y -548.039,Z 1021.008,A 0.000,B 0.000,C 90.000,E1 37.397} C_DIS
LIN {X -0.334,Y -544.195,Z 1021.003,A 0.000,B 0.000,C 90.000,E1 36.583} C_DIS
LIN {X -0.067,Y -539.370,Z 1020.998,A 0.000,B 0.000,C 90.000,E1 35.564} C_DIS
LIN {X 0.255,Y -534.176,Z 1020.992,A 0.000,B 0.000,C 90.000,E1 34.532} C_DIS
LIN {X -0.069,Y -529.346,Z 1020.987,A 0.000,B 0.000,C 90.000,E1 33.706} C_DIS
LIN {X 0.322,Y -525.942,Z 1020.984,A 0.000,B 0.000,C 90.000,E1 33.086} C_DIS
LIN {X -0.088,Y -520.584,Z 1020.979,A 0.000,B 0.000,C 90.000,E1 32.260} C_DIS
LIN {X -0.212,Y -515.766,Z 1020.975,A 0.000,B 0.000,C 90.000,E1 31.544} C_DIS
LIN {X 0.068,Y -511.562,Z 1020.972,A 0.000,B 0.000,C 90.000,E1 30.924} C_DIS
LIN {X 0.052,Y -507.118,Z 1020.969,A 0.000,B 0.000,C 90.000,E1 30.335} C_DIS
LIN {X 0.065,Y -501.088,Z 1020.964,A 0.000,B 0.000,C 90.000,E1 29.589} C_DIS
LIN {X -0.116,Y -494.442,Z 1020.960,A 0.000,B 0.000,C 90.000,E1 28.871} C_DIS
LIN {X -0.086,Y -489.021,Z 1020.957,A 0.000,B 0.000,C 90.000,E1 28.281} C_DIS
LIN {X -0.149,Y -483.342,Z 1020.954,A 0.000,B 0.000,C 90.000,E1 27.719} C_DIS
LIN {X 0.076,Y -472.198,Z 1020.948,A 0.000,B 0.000,C 90.000,E1 26.616} C_DIS
LIN {X -0.251,Y -464.822,Z 1020.944,A 0.000,B 0.000,C 90.000,E1 25.976} C_DIS
LIN {X -0.002,Y -455.778,Z 1020.940,A 0.000,B 0.000,C 90.000,E1 25.155} C_DIS
LIN {X -0.085,Y -449.674,Z 1020.937,A 0.000,B 0.000,C 90.000,E1 24.643} C_DIS
LIN {X 0.001,Y -427.051,Z 1020.926,A 0.000,B 0.000,C 90.000,E1 22.642} C_DIS
LIN {X 0.083,Y -415.319,Z 1020.919,A 0.000,B 0.000,C 90.000,E1 21.482} C_DIS
LIN {X 0.073,Y -401.139,Z 1020.911,A 0.000,B 0.000,C 90.000,E1 19.939} C_DIS
LIN {X 0.181,Y -398.823,Z 1020.909,A 0.000,B 0.000,C 90.000,E1 19.631} C_DIS
LIN {X -0.109,Y -394.829,Z 1020.906,A 0.000,B 0.000,C 90.000,E1 19.087} C_DIS
LIN {X -0.080,Y -392.806,Z 1020.904,A 0.000,B 0.000,C 90.000,E1 18.725} C_DIS
LIN {X 0.213,Y -391.876,Z 1020.903,A 0.000,B 0.000,C 90.000,E1 18.417} C_DIS
LIN {X -0.132,Y -391.472,Z 1020.902,A 0.000,B 0.000,C 90.000,E1 18.290} C_DIS
LIN {X 0.115,Y -390.966,Z 1020.898,A 0.000,B 0.000,C 90.000,E1 17.528} C_DIS
LIN {X 0.030,Y -391.398,Z 1020.892,A 0.000,B 0.000,C 90.000,E1 16.622} C_DIS
LIN {X 0.056,Y -397.008,Z 1020.865,A 0.000,B 0.000,C 90.000,E1 11.658} C_DIS
LIN {X -0.114,Y -404.523,Z 1020.840,A 0.000,B 0.000,C 90.000,E1 7.125} C_DIS
LIN {X -0.164,Y -411.079,Z 1020.822,A 0.000,B 0.000,C 90.000,E1 4.012} C_DIS
LIN {X -0.163,Y -414.203,Z 1020.815,A 0.000,B 0.000,C 90.000,E1 2.636} C_DIS
LIN {X -0.150,Y -416.356,Z 1020.811,A 0.000,B 0.000,C 90.000,E1 1.949} C_DIS
LIN {X -0.131,Y -417.025,Z 1020.810,A 0.000,B 0.000,C 90.000,E1 1.776} C_DIS
LIN {X -0.124,Y -418.000,Z 1020.809,A 0.000,B 0.000,C 90.000,E1 1.604} C_DIS
LIN {X 0.128,Y -422.398,Z 1020.806,A 0.000,B 0.000,C 90.000,E1 0.974} C_DIS
LIN {X -0.075,Y -423.208,Z 1020.805,A 0.000,B 0.000,C 90.000,E1 0.917} C_DIS
LIN {X -0.109,Y -427.646,Z 1020.803,A 0.000,B 0.000,C 90.000,E1 0.573} C_DIS
LIN {X -0.011,Y -435.254,Z 1020.801,A 0.000,B 0.000,C 90.000,E1 0.115} C_DIS
LIN {X 0.148,Y -452.045,Z 1020.795,A 0.000,B 0.000,C 90.000,E1 359.083} C_DIS
LIN {X -0.071,Y -465.077,Z 1020.791,A 0.000,B 0.000,C 90.000,E1 358.339} C_DIS
LIN {X 0.239,Y -479.934,Z 1020.786,A 0.000,B 0.000,C 90.000,E1 357.421} C_DIS
LIN {X 0.162,Y -489.830,Z 1020.783,A 0.000,B 0.000,C 90.000,E1 356.849} C_DIS
LIN {X 0.044,Y -499.466,Z 1020.779,A 0.000,B 0.000,C 90.000,E1 356.274} C_DIS
LIN {X 0.190,Y -509.067,Z 1020.776,A 0.000,B 0.000,C 90.000,E1 355.641} C_DIS
LIN {X 0.214,Y -518.058,Z 1020.772,A 0.000,B 0.000,C 90.000,E1 355.008} C_DIS
LIN {X -0.222,Y -525.492,Z 1020.769,A 0.000,B 0.000,C 90.000,E1 354.489} C_DIS
LIN {X 0.099,Y -534.025,Z 1020.765,A 0.000,B 0.000,C 90.000,E1 353.742} C_DIS
LIN {X 0.170,Y -540.862,Z 1020.762,A 0.000,B 0.000,C 90.000,E1 353.109} C_DIS
LIN {X 0.138,Y -546.042,Z 1020.759,A 0.000,B 0.000,C 90.000,E1 352.591} C_DIS
LIN {X 0.192,Y -552.175,Z 1020.755,A 0.000,B 0.000,C 90.000,E1 351.894} C_DIS
LIN {X -0.186,Y -556.792,Z 1020.752,A 0.000,B 0.000,C 90.000,E1 351.376} C_DIS
LIN {X -0.150,Y -561.847,Z 1020.748,A 0.000,B 0.000,C 90.000,E1 350.679} C_DIS
LIN {X -0.085,Y -566.437,Z 1020.744,A 0.000,B 0.000,C 90.000,E1 349.982} C_DIS
LIN {X 0.261,Y -569.772,Z 1020.741,A 0.000,B 0.000,C 90.000,E1 349.398} C_DIS
LIN {X 0.270,Y -574.502,Z 1020.737,A 0.000,B 0.000,C 90.000,E1 348.578} C_DIS
LIN {X -0.119,Y -578.073,Z 1020.733,A 0.000,B 0.000,C 90.000,E1 347.937} C_DIS
LIN {X -0.026,Y -582.092,Z 1020.728,A 0.000,B 0.000,C 90.000,E1 347.117} C_DIS
LIN {X -0.078,Y -587.033,Z 1020.722,A 0.000,B 0.000,C 90.000,E1 346.047} C_DIS
LIN {X 0.047,Y -592.806,Z 1020.715,A 0.000,B 0.000,C 90.000,E1 344.700} C_DIS
LIN {X 0.135,Y -597.185,Z 1020.709,A 0.000,B 0.000,C 90.000,E1 343.630} C_DIS
LIN {X -0.114,Y -601.413,Z 1020.703,A 0.000,B 0.000,C 90.000,E1 342.598} C_DIS
LIN {X 0.074,Y -603.423,Z 1020.700,A 0.000,B 0.000,C 90.000,E1 342.054} C_DIS
LIN {X -0.274,Y -607.302,Z 1020.695,A 0.000,B 0.000,C 90.000,E1 341.040} C_DIS
LIN {X -0.048,Y -609.120,Z 1020.692,A 0.000,B 0.000,C 90.000,E1 340.496} C_DIS
LIN {X -0.183,Y -613.211,Z 1020.684,A 0.000,B 0.000,C 90.000,E1 339.209} C_DIS
LIN {X 0.011,Y -616.284,Z 1020.679,A 0.000,B 0.000,C 90.000,E1 338.156} C_DIS
LIN {X 0.252,Y -619.115,Z 1020.673,A 0.000,B 0.000,C 90.000,E1 337.102} C_DIS
LIN {X -0.031,Y -621.186,Z 1020.669,A 0.000,B 0.000,C 90.000,E1 336.357} C_DIS
LIN {X -0.300,Y -623.692,Z 1020.663,A 0.000,B 0.000,C 90.000,E1 335.357} C_DIS
LIN {X 0.292,Y -626.004,Z 1020.657,A 0.000,B 0.000,C 90.000,E1 334.280} C_DIS
LIN {X -0.163,Y -629.012,Z 1020.649,A 0.000,B 0.000,C 90.000,E1 332.794} C_DIS
LIN {X -0.089,Y -630.394,Z 1020.645,A 0.000,B 0.000,C 90.000,E1 332.025} C_DIS
LIN {X -0.157,Y -632.815,Z 1020.636,A 0.000,B 0.000,C 90.000,E1 330.511} C_DIS
LIN {X -0.024,Y -634.270,Z 1020.631,A 0.000,B 0.000,C 90.000,E1 329.488} C_DIS
LIN {X 0.257,Y -635.791,Z 1020.624,A 0.000,B 0.000,C 90.000,E1 328.201} C_DIS
LIN {X -0.433,Y -637.547,Z 1020.614,A 0.000,B 0.000,C 90.000,E1 326.501} C_DIS
LIN {X -0.131,Y -638.344,Z 1020.608,A 0.000,B 0.000,C 90.000,E1 325.468} C_DIS
LIN {X -0.343,Y -638.859,Z 1020.603,A 0.000,B 0.000,C 90.000,E1 324.482} C_DIS
LIN {X 0.345,Y -639.246,Z 1020.597,A 0.000,B 0.000,C 90.000,E1 323.417} C_DIS
LIN {X 0.031,Y -639.572,Z 1020.590,A 0.000,B 0.000,C 90.000,E1 322.190} C_DIS
LIN {X 0.112,Y -639.873,Z 1020.582,A 0.000,B 0.000,C 90.000,E1 320.678} C_DIS
LIN {X 0.012,Y -640.482,Z 1020.572,A 0.000,B 0.000,C 90.000,E1 318.933} C_DIS
LIN {X 0.227,Y -640.894,Z 1020.568,A 0.000,B 0.000,C 90.000,E1 318.162} C_DIS
LIN {X -0.323,Y -641.499,Z 1020.558,A 0.000,B 0.000,C 90.000,E1 316.458} C_DIS
LIN {X 0.028,Y -642.290,Z 1020.548,A 0.000,B 0.000,C 90.000,E1 314.676} C_DIS
LIN {X 0.107,Y -642.901,Z 1020.541,A 0.000,B 0.000,C 90.000,E1 313.419} C_DIS
LIN {X 0.199,Y -643.522,Z 1020.534,A 0.000,B 0.000,C 90.000,E1 312.162} C_DIS
LIN {X -0.210,Y -644.078,Z 1020.526,A 0.000,B 0.000,C 90.000,E1 310.701} C_DIS
LIN {X -0.046,Y -644.397,Z 1020.521,A 0.000,B 0.000,C 90.000,E1 309.688} C_DIS
LIN {X 0.131,Y -644.890,Z 1020.512,A 0.000,B 0.000,C 90.000,E1 308.177} C_DIS
LIN {X 0.393,Y -645.061,Z 1020.507,A 0.000,B 0.000,C 90.000,E1 307.156} C_DIS
LIN {X 0.105,Y -645.432,Z 1020.497,A 0.000,B 0.000,C 90.000,E1 305.438} C_DIS
LIN {X -0.023,Y -646.167,Z 1020.483,A 0.000,B 0.000,C 90.000,E1 302.959} C_DIS
LIN {X 0.266,Y -649.016,Z 1020.462,A 0.000,B 0.000,C 90.000,E1 299.205} C_DIS
LIN {X -0.226,Y -650.895,Z 1020.453,A 0.000,B 0.000,C 90.000,E1 297.513} C_DIS
LIN {X 0.276,Y -652.277,Z 1020.446,A 0.000,B 0.000,C 90.000,E1 296.232} C_DIS
LIN {X -0.177,Y -653.200,Z 1020.440,A 0.000,B 0.000,C 90.000,E1 295.283} C_DIS
LIN {X 0.142,Y -653.649,Z 1020.436,A 0.000,B 0.000,C 90.000,E1 294.515} C_DIS
LIN {X 0.194,Y -653.917,Z 1020.432,A 0.000,B 0.000,C 90.000,E1 293.770} C_DIS
LIN {X -0.245,Y -653.969,Z 1020.427,A 0.000,B 0.000,C 90.000,E1 292.823} C_DIS
LIN {X -0.334,Y -653.816,Z 1020.421,A 0.000,B 0.000,C 90.000,E1 291.844} C_DIS
LIN {X -0.139,Y -653.165,Z 1020.419,A 0.000,B 0.000,C 90.000,E1 291.334} C_DIS
LIN {X -0.280,Y -652.684,Z 1020.417,A 0.000,B 0.000,C 90.000,E1 291.099} C_DIS
LIN {X -0.327,Y -651.228,Z 1020.414,A 0.000,B 0.000,C 90.000,E1 290.610} C_DIS
LIN {X -0.284,Y -650.701,Z 1020.414,A 0.000,B 0.000,C 90.000,E1 290.482} C_DIS
LIN {X 0.368,Y -649.840,Z 1020.413,A 0.000,B 0.000,C 90.000,E1 290.301} C_DIS
LIN {X 0.184,Y -648.771,Z 1020.412,A 0.000,B 0.000,C 90.000,E1 290.194} C_DIS
LIN {X 0.296,Y -646.043,Z 1020.410,A 0.000,B 0.000,C 90.000,E1 289.812} C_DIS
LIN {X 0.110,Y -644.623,Z 1020.410,A 0.000,B 0.000,C 90.000,E1 289.704} C_DIS
LIN {X 0.143,Y -642.667,Z 1020.409,A 0.000,B 0.000,C 90.000,E1 289.577} C_DIS
LIN {X -0.116,Y -638.982,Z 1020.407,A 0.000,B 0.000,C 90.000,E1 289.322} C_DIS
LIN {X -0.084,Y -637.182,Z 1020.407,A 0.000,B 0.000,C 90.000,E1 289.214} C_DIS
LIN {X 0.122,Y -630.414,Z 1020.405,A 0.000,B 0.000,C 90.000,E1 288.852} C_DIS
LIN {X 0.041,Y -619.958,Z 1020.402,A 0.000,B 0.000,C 90.000,E1 288.417} C_DIS
LIN {X -0.146,Y -616.516,Z 1020.402,A 0.000,B 0.000,C 90.000,E1 288.308} C_DIS
LIN {X -0.195,Y -616.411,Z 1020.402,A 0.000,B 0.000,C 90.000,E1 288.308} C_DIS
LIN {X 0.309,Y -616.227,Z 1020.401,A 0.000,B 0.000,C 90.000,E1 288.236} C_DIS
LIN {X 0.266,Y -616.230,Z 1020.401,A 0.000,B 0.000,C 90.000,E1 288.236} C_DIS
LIN {X 0.223,Y -616.802,Z 1020.401,A 0.000,B 0.000,C 90.000,E1 288.127} C_DIS
LIN {X 0.176,Y -618.704,Z 1020.399,A 0.000,B 0.000,C 90.000,E1 287.873} C_DIS
LIN {X -0.082,Y -621.899,Z 1020.397,A 0.000,B 0.000,C 90.000,E1 287.511} C_DIS
LIN {X 0.071,Y -625.909,Z 1020.394,A 0.000,B 0.000,C 90.000,E1 286.985} C_DIS
LIN {X -0.174,Y -630.390,Z 1020.391,A 0.000,B 0.000,C 90.000,E1 286.370} C_DIS
LIN {X 0.037,Y -634.079,Z 1020.387,A 0.000,B 0.000,C 90.000,E1 285.717} C_DIS
LIN {X 0.112,Y -637.612,Z 1020.383,A 0.000,B 0.000,C 90.000,E1 284.954} C_DIS
LIN {X -0.061,Y -638.658,Z 1020.382,A 0.000,B 0.000,C 90.000,E1 284.717} C_DIS
LIN {X 0.226,Y -640.337,Z 1020.379,A 0.000,B 0.000,C 90.000,E1 284.189} C_DIS
LIN {X 0.057,Y -641.845,Z 1020.376,A 0.000,B 0.000,C 90.000,E1 283.703} C_DIS
LIN {X 0.366,Y -642.804,Z 1020.373,A 0.000,B 0.000,C 90.000,E1 283.175} C_DIS
LIN {X -0.238,Y -643.660,Z 1020.369,A 0.000,B 0.000,C 90.000,E1 282.479} C_DIS
LIN {X 0.091,Y -643.985,Z 1020.367,A 0.000,B 0.000,C 90.000,E1 281.951} C_DIS
LIN {X -0.212,Y -643.944,Z 1020.364,A 0.000,B 0.000,C 90.000,E1 281.478} C_DIS
LIN {X 0.114,Y -643.480,Z 1020.361,A 0.000,B 0.000,C 90.000,E1 280.950} C_DIS
LIN {X -0.041,Y -643.171,Z 1020.360,A 0.000,B 0.000,C 90.000,E1 280.715} C_DIS
LIN {X 0.162,Y -642.217,Z 1020.357,A 0.000,B 0.000,C 90.000,E1 280.197} C_DIS
LIN {X -0.159,Y -640.874,Z 1020.354,A 0.000,B 0.000,C 90.000,E1 279.726} C_DIS
LIN {X 0.035,Y -639.169,Z 1020.351,A 0.000,B 0.000,C 90.000,E1 279.208} C_DIS
LIN {X -0.135,Y -638.144,Z 1020.350,A 0.000,B 0.000,C 90.000,E1 278.973} C_DIS
LIN {X 0.042,Y -635.624,Z 1020.347,A 0.000,B 0.000,C 90.000,E1 278.454} C_DIS
LIN {X 0.204,Y -632.538,Z 1020.344,A 0.000,B 0.000,C 90.000,E1 277.936} C_DIS
LIN {X -0.195,Y -628.879,Z 1020.341,A 0.000,B 0.000,C 90.000,E1 277.466} C_DIS
LIN {X -0.230,Y -623.124,Z 1020.338,A 0.000,B 0.000,C 90.000,E1 276.834} C_DIS
LIN {X 0.062,Y -619.119,Z 1020.336,A 0.000,B 0.000,C 90.000,E1 276.429} C_DIS
LIN {X -0.004,Y -613.653,Z 1020.333,A 0.000,B 0.000,C 90.000,E1 275.967} C_DIS
LIN {X 0.054,Y -609.061,Z 1020.331,A 0.000,B 0.000,C 90.000,E1 275.625} C_DIS
LIN {X -0.203,Y -604.354,Z 1020.330,A 0.000,B 0.000,C 90.000,E1 275.334} C_DIS
LIN {X -0.214,Y -599.649,Z 1020.328,A 0.000,B 0.000,C 90.000,E1 275.049} C_DIS
LIN {X -0.152,Y -592.940,Z 1020.326,A 0.000,B 0.000,C 90.000,E1 274.702} C_DIS
LIN {X -0.184,Y -585.667,Z 1020.324,A 0.000,B 0.000,C 90.000,E1 274.416} C_DIS
LIN {X -0.085,Y -577.850,Z 1020.323,A 0.000,B 0.000,C 90.000,E1 274.188} C_DIS
LIN {X -0.195,Y -571.659,Z 1020.323,A 0.000,B 0.000,C 90.000,E1 274.069} C_DIS
LIN {X 0.242,Y -566.768,Z 1020.322,A 0.000,B 0.000,C 90.000,E1 273.955} C_DIS
LIN {X -0.005,Y -563.645,Z 1020.322,A 0.000,B 0.000,C 90.000,E1 273.955} C_DIS
LIN {X -0.149,Y -559.292,Z 1020.322,A 0.000,B 0.000,C 90.000,E1 273.955} C_DIS
LIN {X -0.179,Y -544.011,Z 1020.322,A 0.000,B 0.000,C 90.000,E1 273.955} C_DIS
LIN {X 0.002,Y -543.491,Z 1020.321,A 0.000,B 0.000,C 90.000,E1 273.841} C_DIS
LIN {X -0.254,Y -543.209,Z 1020.321,A 0.000,B 0.000,C 90.000,E1 273.784} C_DIS
LIN {X 0.026,Y -542.095,Z 1020.317,A 0.000,B 0.000,C 90.000,E1 273.037} C_DIS
LIN {X -0.266,Y -540.453,Z 1020.301,A 0.000,B 0.000,C 90.000,E1 270.229} C_DIS
LIN {X -0.182,Y -539.736,Z 1020.295,A 0.000,B 0.000,C 90.000,E1 269.083} C_DIS
LIN {X -0.098,Y -538.851,Z 1020.289,A 0.000,B 0.000,C 90.000,E1 267.936} C_DIS
LIN {X -0.011,Y -537.785,Z 1020.281,A 0.000,B 0.000,C 90.000,E1 266.502} C_DIS
LIN {X 0.087,Y -536.512,Z 1020.271,A 0.000,B 0.000,C 90.000,E1 264.780} C_DIS
LIN {X 0.212,Y -535.380,Z 1020.263,A 0.000,B 0.000,C 90.000,E1 263.337} C_DIS
LIN {X -0.259,Y -534.469,Z 1020.257,A 0.000,B 0.000,C 90.000,E1 262.243} C_DIS
LIN {X -0.145,Y -533.285,Z 1020.250,A 0.000,B 0.000,C 90.000,E1 261.084} C_DIS
LIN {X -0.051,Y -531.957,Z 1020.244,A 0.000,B 0.000,C 90.000,E1 259.926} C_DIS
LIN {X 0.226,Y -529.731,Z 1020.233,A 0.000,B 0.000,C 90.000,E1 257.881} C_DIS
LIN {X -0.009,Y -528.226,Z 1020.225,A 0.000,B 0.000,C 90.000,E1 256.464} C_DIS
LIN {X 0.243,Y -526.580,Z 1020.217,A 0.000,B 0.000,C 90.000,E1 254.991} C_DIS
LIN {X 0.092,Y -524.966,Z 1020.209,A 0.000,B 0.000,C 90.000,E1 253.559} C_DIS
LIN {X 0.066,Y -523.122,Z 1020.199,A 0.000,B 0.000,C 90.000,E1 251.819} C_DIS
LIN {X -0.128,Y -522.107,Z 1020.194,A 0.000,B 0.000,C 90.000,E1 250.967} C_DIS
LIN {X -0.206,Y -520.239,Z 1020.186,A 0.000,B 0.000,C 90.000,E1 249.518} C_DIS
LIN {X 0.046,Y -518.312,Z 1020.178,A 0.000,B 0.000,C 90.000,E1 248.028} C_DIS
LIN {X 0.062,Y -515.559,Z 1020.167,A 0.000,B 0.000,C 90.000,E1 245.973} C_DIS
LIN {X 0.092,Y -512.936,Z 1020.157,A 0.000,B 0.000,C 90.000,E1 244.204} C_DIS
LIN {X -0.050,Y -510.655,Z 1020.149,A 0.000,B 0.000,C 90.000,E1 242.743} C_DIS
LIN {X -0.048,Y -507.138,Z 1020.137,A 0.000,B 0.000,C 90.000,E1 240.667} C_DIS
LIN {X 0.107,Y -505.072,Z 1020.130,A 0.000,B 0.000,C 90.000,E1 239.459} C_DIS
LIN {X -0.072,Y -503.409,Z 1020.125,A 0.000,B 0.000,C 90.000,E1 238.584} C_DIS
LIN {X -0.068,Y -499.930,Z 1020.115,A 0.000,B 0.000,C 90.000,E1 236.786} C_DIS
LIN {X -0.024,Y -495.966,Z 1020.105,A 0.000,B 0.000,C 90.000,E1 234.975} C_DIS
LIN {X 0.218,Y -491.631,Z 1020.095,A 0.000,B 0.000,C 90.000,E1 233.130} C_DIS
LIN {X 0.131,Y -487.957,Z 1020.087,A 0.000,B 0.000,C 90.000,E1 231.618} C_DIS
LIN {X 0.096,Y -483.734,Z 1020.077,A 0.000,B 0.000,C 90.000,E1 229.784} C_DIS
LIN {X 0.143,Y -478.184,Z 1020.063,A 0.000,B 0.000,C 90.000,E1 227.310} C_DIS
LIN {X 0.109,Y -472.395,Z 1020.047,A 0.000,B 0.000,C 90.000,E1 224.514} C_DIS
LIN {X 0.146,Y -467.160,Z 1020.034,A 0.000,B 0.000,C 90.000,E1 222.000} C_DIS
LIN {X -0.151,Y -463.941,Z 1020.025,A 0.000,B 0.000,C 90.000,E1 220.458} C_DIS
LIN {X -0.201,Y -461.187,Z 1020.018,A 0.000,B 0.000,C 90.000,E1 219.197} C_DIS
LIN {X 0.067,Y -458.316,Z 1020.011,A 0.000,B 0.000,C 90.000,E1 217.890} C_DIS
LIN {X -0.093,Y -451.943,Z 1019.995,A 0.000,B 0.000,C 90.000,E1 215.025} C_DIS
LIN {X -0.096,Y -447.716,Z 1019.984,A 0.000,B 0.000,C 90.000,E1 213.086} C_DIS
LIN {X -0.125,Y -444.158,Z 1019.975,A 0.000,B 0.000,C 90.000,E1 211.465} C_DIS
LIN {X 0.102,Y -441.398,Z 1019.968,A 0.000,B 0.000,C 90.000,E1 210.129} C_DIS
LIN {X 0.101,Y -437.683,Z 1019.958,A 0.000,B 0.000,C 90.000,E1 208.487} C_DIS
LIN {X 0.042,Y -432.412,Z 1019.946,A 0.000,B 0.000,C 90.000,E1 206.181} C_DIS
LIN {X 0.220,Y -427.154,Z 1019.933,A 0.000,B 0.000,C 90.000,E1 203.823} C_DIS
LIN {X -0.052,Y -422.709,Z 1019.921,A 0.000,B 0.000,C 90.000,E1 201.844} C_DIS
LIN {X -0.097,Y -417.441,Z 1019.906,A 0.000,B 0.000,C 90.000,E1 199.141} C_DIS
LIN {X -0.184,Y -412.084,Z 1019.889,A 0.000,B 0.000,C 90.000,E1 196.079} C_DIS
LIN {X -0.001,Y -408.009,Z 1019.874,A 0.000,B 0.000,C 90.000,E1 193.300} C_DIS
LIN {X -0.154,Y -405.822,Z 1019.864,A 0.000,B 0.000,C 90.000,E1 191.591} C_DIS
LIN {X -0.127,Y -404.818,Z 1019.859,A 0.000,B 0.000,C 90.000,E1 190.546} C_DIS
LIN {X -0.113,Y -404.579,Z 1019.855,A 0.000,B 0.000,C 90.000,E1 189.849} C_DIS
LIN {X -0.107,Y -404.703,Z 1019.853,A 0.000,B 0.000,C 90.000,E1 189.500} C_DIS
LIN {X -0.053,Y -405.621,Z 1019.849,A 0.000,B 0.000,C 90.000,E1 188.803} C_DIS
LIN {X -0.046,Y -405.993,Z 1019.847,A 0.000,B 0.000,C 90.000,E1 188.454} C_DIS
LIN {X -0.105,Y -408.275,Z 1019.843,A 0.000,B 0.000,C 90.000,E1 187.757} C_DIS
LIN {X -0.107,Y -410.407,Z 1019.840,A 0.000,B 0.000,C 90.000,E1 187.239} C_DIS
LIN {X -0.149,Y -414.863,Z 1019.836,A 0.000,B 0.000,C 90.000,E1 186.429} C_DIS
LIN {X -0.005,Y -422.141,Z 1019.830,A 0.000,B 0.000,C 90.000,E1 185.391} C_DIS
LIN {X -0.056,Y -429.907,Z 1019.825,A 0.000,B 0.000,C 90.000,E1 184.416} C_DIS
LIN {X 0.173,Y -443.410,Z 1019.815,A 0.000,B 0.000,C 90.000,E1 182.751} C_DIS
LIN {X 0.204,Y -455.222,Z 1019.807,A 0.000,B 0.000,C 90.000,E1 181.318} C_DIS
LIN {X -0.040,Y -464.060,Z 1019.801,A 0.000,B 0.000,C 90.000,E1 180.229} C_DIS
LIN {X -0.059,Y -473.747,Z 1019.794,A 0.000,B 0.000,C 90.000,E1 178.969} C_DIS
LIN {X -0.203,Y -480.711,Z 1019.789,A 0.000,B 0.000,C 90.000,E1 178.051} C_DIS
LIN {X 0.198,Y -487.462,Z 1019.784,A 0.000,B 0.000,C 90.000,E1 177.078} C_DIS
LIN {X -0.112,Y -494.930,Z 1019.778,A 0.000,B 0.000,C 90.000,E1 176.045} C_DIS
LIN {X -0.108,Y -502.965,Z 1019.771,A 0.000,B 0.000,C 90.000,E1 174.837} C_DIS
LIN {X -0.179,Y -509.714,Z 1019.766,A 0.000,B 0.000,C 90.000,E1 173.799} C_DIS
LIN {X -0.164,Y -516.255,Z 1019.760,A 0.000,B 0.000,C 90.000,E1 172.761} C_DIS
LIN {X 0.163,Y -526.487,Z 1019.750,A 0.000,B 0.000,C 90.000,E1 170.971} C_DIS
LIN {X 0.147,Y -539.007,Z 1019.738,A 0.000,B 0.000,C 90.000,E1 168.814} C_DIS
LIN {X 0.085,Y -544.720,Z 1019.732,A 0.000,B 0.000,C 90.000,E1 167.825} C_DIS
LIN {X 0.055,Y -551.053,Z 1019.726,A 0.000,B 0.000,C 90.000,E1 166.700} C_DIS
LIN {X 0.258,Y -558.735,Z 1019.718,A 0.000,B 0.000,C 90.000,E1 165.283} C_DIS
LIN {X 0.053,Y -566.239,Z 1019.711,A 0.000,B 0.000,C 90.000,E1 163.921} C_DIS
LIN {X -0.047,Y -571.880,Z 1019.705,A 0.000,B 0.000,C 90.000,E1 162.834} C_DIS
LIN {X -0.241,Y -577.240,Z 1019.699,A 0.000,B 0.000,C 90.000,E1 161.764} C_DIS
LIN {X -0.268,Y -582.933,Z 1019.692,A 0.000,B 0.000,C 90.000,E1 160.550} C_DIS
LIN {X -0.215,Y -588.193,Z 1019.685,A 0.000,B 0.000,C 90.000,E1 159.337} C_DIS
LIN {X 0.183,Y -592.623,Z 1019.679,A 0.000,B 0.000,C 90.000,E1 158.230} C_DIS
LIN {X -0.359,Y -595.789,Z 1019.675,A 0.000,B 0.000,C 90.000,E1 157.486} C_DIS
LIN {X -0.086,Y -598.715,Z 1019.670,A 0.000,B 0.000,C 90.000,E1 156.666} C_DIS
LIN {X -0.095,Y -602.377,Z 1019.664,A 0.000,B 0.000,C 90.000,E1 155.613} C_DIS
LIN {X 0.193,Y -605.710,Z 1019.659,A 0.000,B 0.000,C 90.000,E1 154.537} C_DIS
LIN {X 0.031,Y -608.132,Z 1019.654,A 0.000,B 0.000,C 90.000,E1 153.768} C_DIS
LIN {X -0.186,Y -611.862,Z 1019.647,A 0.000,B 0.000,C 90.000,E1 152.487} C_DIS
LIN {X 0.001,Y -614.024,Z 1019.643,A 0.000,B 0.000,C 90.000,E1 151.691} C_DIS
LIN {X 0.155,Y -618.081,Z 1019.634,A 0.000,B 0.000,C 90.000,E1 150.127} C_DIS
LIN {X 0.154,Y -622.708,Z 1019.624,A 0.000,B 0.000,C 90.000,E1 148.329} C_DIS
LIN {X -0.078,Y -625.345,Z 1019.618,A 0.000,B 0.000,C 90.000,E1 147.327} C_DIS
LIN {X 0.406,Y -628.559,Z 1019.611,A 0.000,B 0.000,C 90.000,E1 146.008} C_DIS
LIN {X -0.078,Y -632.965,Z 1019.602,A 0.000,B 0.000,C 90.000,E1 144.276} C_DIS
LIN {X 0.020,Y -635.526,Z 1019.596,A 0.000,B 0.000,C 90.000,E1 143.256} C_DIS
LIN {X 0.162,Y -638.642,Z 1019.589,A 0.000,B 0.000,C 90.000,E1 141.984} C_DIS
LIN {X -0.260,Y -642.342,Z 1019.581,A 0.000,B 0.000,C 90.000,E1 140.517} C_DIS
LIN {X 0.378,Y -644.755,Z 1019.575,A 0.000,B 0.000,C 90.000,E1 139.461} C_DIS
LIN {X 0.070,Y -647.786,Z 1019.568,A 0.000,B 0.000,C 90.000,E1 138.243} C_DIS
LIN {X -0.354,Y -652.765,Z 1019.557,A 0.000,B 0.000,C 90.000,E1 136.296} C_DIS
LIN {X 0.363,Y -656.145,Z 1019.550,A 0.000,B 0.000,C 90.000,E1 135.000} C_DIS
LIN {X -0.330,Y -662.716,Z 1019.538,A 0.000,B 0.000,C 90.000,E1 132.852} C_DIS
LIN {X 0.107,Y -665.788,Z 1019.533,A 0.000,B 0.000,C 90.000,E1 131.838} C_DIS
LIN {X 0.145,Y -668.741,Z 1019.527,A 0.000,B 0.000,C 90.000,E1 130.862} C_DIS
LIN {X -0.289,Y -671.631,Z 1019.522,A 0.000,B 0.000,C 90.000,E1 129.930} C_DIS
LIN {X -0.063,Y -675.735,Z 1019.514,A 0.000,B 0.000,C 90.000,E1 128.463} C_DIS
LIN {X 0.230,Y -679.043,Z 1019.507,A 0.000,B 0.000,C 90.000,E1 127.237} C_DIS
LIN {X 0.192,Y -682.900,Z 1019.499,A 0.000,B 0.000,C 90.000,E1 125.804} C_DIS
LIN {X 0.198,Y -686.125,Z 1019.492,A 0.000,B 0.000,C 90.000,E1 124.612} C_DIS
LIN {X 0.033,Y -687.981,Z 1019.488,A 0.000,B 0.000,C 90.000,E1 123.913} C_DIS
LIN {X -0.047,Y -691.581,Z 1019.481,A 0.000,B 0.000,C 90.000,E1 122.498} C_DIS
LIN {X -0.290,Y -694.521,Z 1019.474,A 0.000,B 0.000,C 90.000,E1 121.337} C_DIS
LIN {X 0.099,Y -697.124,Z 1019.467,A 0.000,B 0.000,C 90.000,E1 120.129} C_DIS
LIN {X 0.263,Y -698.473,Z 1019.464,A 0.000,B 0.000,C 90.000,E1 119.411} C_DIS
LIN {X 0.364,Y -700.232,Z 1019.457,A 0.000,B 0.000,C 90.000,E1 118.231} C_DIS
LIN {X -0.062,Y -701.046,Z 1019.453,A 0.000,B 0.000,C 90.000,E1 117.564} C_DIS
LIN {X -0.088,Y -702.813,Z 1019.441,A 0.000,B 0.000,C 90.000,E1 115.463} C_DIS
LIN {X -0.182,Y -703.299,Z 1019.438,A 0.000,B 0.000,C 90.000,E1 114.771} C_DIS
LIN {X 0.090,Y -703.296,Z 1019.435,A 0.000,B 0.000,C 90.000,E1 114.283} C_DIS
LIN {X -0.271,Y -703.186,Z 1019.434,A 0.000,B 0.000,C 90.000,E1 114.079} C_DIS
LIN {X 0.005,Y -702.444,Z 1019.431,A 0.000,B 0.000,C 90.000,E1 113.590} C_DIS
LIN {X 0.282,Y -701.705,Z 1019.430,A 0.000,B 0.000,C 90.000,E1 113.334} C_DIS
LIN {X -0.093,Y -699.130,Z 1019.427,A 0.000,B 0.000,C 90.000,E1 112.898} C_DIS
LIN {X 0.039,Y -698.332,Z 1019.427,A 0.000,B 0.000,C 90.000,E1 112.770} C_DIS
LIN {X 0.170,Y -697.146,Z 1019.426,A 0.000,B 0.000,C 90.000,E1 112.642} C_DIS
LIN {X -0.007,Y -692.032,Z 1019.424,A 0.000,B 0.000,C 90.000,E1 112.333} C_DIS
LIN {X -0.193,Y -690.573,Z 1019.424,A 0.000,B 0.000,C 90.000,E1 112.259} C_DIS
LIN {X -0.010,Y -688.788,Z 1019.423,A 0.000,B 0.000,C 90.000,E1 112.153} C_DIS
LIN {X -0.250,Y -684.106,Z 1019.422,A 0.000,B 0.000,C 90.000,E1 112.025} C_DIS
LIN {X -0.158,Y -675.394,Z 1019.422,A 0.000,B 0.000,C 90.000,E1 111.897} C_DIS
LIN {X -0.196,Y -615.387,Z 1019.422,A 0.000,B 0.000,C 90.000,E1 111.897} C_DIS
LIN {X -0.127,Y -610.684,Z 1019.421,A 0.000,B 0.000,C 90.000,E1 111.770} C_DIS
LIN {X -0.133,Y -605.465,Z 1019.420,A 0.000,B 0.000,C 90.000,E1 111.589} C_DIS
LIN {X 0.034,Y -599.135,Z 1019.418,A 0.000,B 0.000,C 90.000,E1 111.280} C_DIS
LIN {X 0.064,Y -593.216,Z 1019.416,A 0.000,B 0.000,C 90.000,E1 110.918} C_DIS
LIN {X -0.251,Y -586.249,Z 1019.413,A 0.000,B 0.000,C 90.000,E1 110.429} C_DIS
LIN {X 0.045,Y -577.972,Z 1019.410,A 0.000,B 0.000,C 90.000,E1 109.704} C_DIS
LIN {X -0.168,Y -571.941,Z 1019.407,A 0.000,B 0.000,C 90.000,E1 109.268} C_DIS
LIN {X -0.001,Y -570.349,Z 1019.406,A 0.000,B 0.000,C 90.000,E1 109.141} C_DIS
LIN {X -0.021,Y -561.852,Z 1019.404,A 0.000,B 0.000,C 90.000,E1 108.671} C_DIS
LIN {X -0.277,Y -555.317,Z 1019.402,A 0.000,B 0.000,C 90.000,E1 108.362} C_DIS
LIN {X 0.025,Y -549.700,Z 1019.400,A 0.000,B 0.000,C 90.000,E1 108.000} C_DIS
LIN {X 0.216,Y -548.380,Z 1019.399,A 0.000,B 0.000,C 90.000,E1 107.819} C_DIS
LIN {X 0.174,Y -548.360,Z 1019.399,A 0.000,B 0.000,C 90.000,E1 107.819} C_DIS
LIN {X 0.172,Y -548.008,Z 1019.397,A 0.000,B 0.000,C 90.000,E1 107.402} C_DIS
LIN {X 0.201,Y -548.220,Z 1019.392,A 0.000,B 0.000,C 90.000,E1 106.567} C_DIS
LIN {X -0.072,Y -548.927,Z 1019.384,A 0.000,B 0.000,C 90.000,E1 105.190} C_DIS
LIN {X -0.020,Y -551.336,Z 1019.364,A 0.000,B 0.000,C 90.000,E1 101.535} C_DIS
LIN {X -0.146,Y -553.944,Z 1019.350,A 0.000,B 0.000,C 90.000,E1 99.029} C_DIS
LIN {X 0.137,Y -554.901,Z 1019.345,A 0.000,B 0.000,C 90.000,E1 98.163} C_DIS
LIN {X 0.247,Y -557.031,Z 1019.335,A 0.000,B 0.000,C 90.000,E1 96.201} C_DIS
LIN {X 0.080,Y -558.088,Z 1019.328,A 0.000,B 0.000,C 90.000,E1 95.106} C_DIS
LIN {X -0.200,Y -558.738,Z 1019.324,A 0.000,B 0.000,C 90.000,E1 94.302} C_DIS
LIN {X -0.271,Y -559.589,Z 1019.316,A 0.000,B 0.000,C 90.000,E1 92.922} C_DIS
LIN {X 0.196,Y -560.215,Z 1019.308,A 0.000,B 0.000,C 90.000,E1 91.489} C_DIS
LIN {X 0.105,Y -560.804,Z 1019.301,A 0.000,B 0.000,C 90.000,E1 90.115} C_DIS
LIN {X 0.120,Y -561.467,Z 1019.292,A 0.000,B 0.000,C 90.000,E1 88.453} C_DIS
LIN {X -0.036,Y -561.825,Z 1019.285,A 0.000,B 0.000,C 90.000,E1 87.364} C_DIS
LIN {X 0.043,Y -562.195,Z 1019.276,A 0.000,B 0.000,C 90.000,E1 85.698} C_DIS
LIN {X 0.269,Y -562.544,Z 1019.265,A 0.000,B 0.000,C 90.000,E1 83.742} C_DIS
LIN {X -0.231,Y -562.848,Z 1019.258,A 0.000,B 0.000,C 90.000,E1 82.413} C_DIS
LIN {X 0.146,Y -563.389,Z 1019.247,A 0.000,B 0.000,C 90.000,E1 80.443} C_DIS
LIN {X 0.071,Y -564.088,Z 1019.236,A 0.000,B 0.000,C 90.000,E1 78.522} C_DIS
LIN {X 0.120,Y -565.128,Z 1019.226,A 0.000,B 0.000,C 90.000,E1 76.589} C_DIS
LIN {X -0.083,Y -566.356,Z 1019.215,A 0.000,B 0.000,C 90.000,E1 74.685} C_DIS
LIN {X -0.246,Y -567.855,Z 1019.204,A 0.000,B 0.000,C 90.000,E1 72.779} C_DIS
LIN {X -0.177,Y -568.811,Z 1019.197,A 0.000,B 0.000,C 90.000,E1 71.402} C_DIS
LIN {X 0.084,Y -569.845,Z 1019.189,A 0.000,B 0.000,C 90.000,E1 70.007} C_DIS
LIN {X -0.003,Y -571.173,Z 1019.178,A 0.000,B 0.000,C 90.000,E1 68.103} C_DIS
LIN {X 0.154,Y -572.265,Z 1019.168,A 0.000,B 0.000,C 90.000,E1 66.177} C_DIS
LIN {X 0.045,Y -573.164,Z 1019.157,A 0.000,B 0.000,C 90.000,E1 64.280} C_DIS
LIN {X -0.141,Y -573.802,Z 1019.148,A 0.000,B 0.000,C 90.000,E1 62.666} C_DIS
LIN {X -0.154,Y -574.329,Z 1019.141,A 0.000,B 0.000,C 90.000,E1 61.307} C_DIS
LIN {X 0.117,Y -574.760,Z 1019.133,A 0.000,B 0.000,C 90.000,E1 59.921} C_DIS
LIN {X -0.097,Y -575.147,Z 1019.125,A 0.000,B 0.000,C 90.000,E1 58.584} C_DIS
LIN {X -0.337,Y -575.629,Z 1019.115,A 0.000,B 0.000,C 90.000,E1 56.707} C_DIS
LIN {X -0.068,Y -575.790,Z 1019.109,A 0.000,B 0.000,C 90.000,E1 55.595} C_DIS
LIN {X 0.356,Y -575.888,Z 1019.101,A 0.000,B 0.000,C 90.000,E1 54.196} C_DIS
LIN {X 0.312,Y -575.698,Z 1019.094,A 0.000,B 0.000,C 90.000,E1 52.844} C_DIS
LIN {X 0.107,Y -575.378,Z 1019.088,A 0.000,B 0.000,C 90.000,E1 51.778} C_DIS
LIN {X -0.196,Y -574.901,Z 1019.082,A 0.000,B 0.000,C 90.000,E1 50.723} C_DIS
LIN {X -0.059,Y -574.274,Z 1019.076,A 0.000,B 0.000,C 90.000,E1 49.622} C_DIS
LIN {X 0.140,Y -573.281,Z 1019.068,A 0.000,B 0.000,C 90.000,E1 48.243} C_DIS
LIN {X -0.318,Y -572.546,Z 1019.064,A 0.000,B 0.000,C 90.000,E1 47.472} C_DIS
LIN {X 0.023,Y -571.653,Z 1019.059,A 0.000,B 0.000,C 90.000,E1 46.620} C_DIS
LIN {X 0.048,Y -570.182,Z 1019.053,A 0.000,B 0.000,C 90.000,E1 45.526} C_DIS
LIN {X -0.052,Y -568.870,Z 1019.048,A 0.000,B 0.000,C 90.000,E1 44.717} C_DIS
LIN {X -0.066,Y -566.849,Z 1019.042,A 0.000,B 0.000,C 90.000,E1 43.623} C_DIS
LIN {X 0.212,Y -565.144,Z 1019.038,A 0.000,B 0.000,C 90.000,E1 42.771} C_DIS
LIN {X 0.053,Y -563.154,Z 1019.033,A 0.000,B 0.000,C 90.000,E1 41.962} C_DIS
LIN {X -0.084,Y -560.934,Z 1019.029,A 0.000,B 0.000,C 90.000,E1 41.148} C_DIS
LIN {X -0.324,Y -559.298,Z 1019.026,A 0.000,B 0.000,C 90.000,E1 40.620} C_DIS
LIN {X -0.135,Y -556.581,Z 1019.021,A 0.000,B 0.000,C 90.000,E1 39.769} C_DIS
LIN {X 0.022,Y -554.667,Z 1019.018,A 0.000,B 0.000,C 90.000,E1 39.197} C_DIS
LIN {X 0.169,Y -552.551,Z 1019.015,A 0.000,B 0.000,C 90.000,E1 38.624} C_DIS
LIN {X -0.130,Y -550.311,Z 1019.012,A 0.000,B 0.000,C 90.000,E1 38.096} C_DIS
LIN {X 0.229,Y -546.038,Z 1019.006,A 0.000,B 0.000,C 90.000,E1 37.076} C_DIS
LIN {X 0.022,Y -542.084,Z 1019.001,A 0.000,B 0.000,C 90.000,E1 36.251} C_DIS
LIN {X 0.245,Y -538.556,Z 1018.997,A 0.000,B 0.000,C 90.000,E1 35.518} C_DIS
LIN {X 0.118,Y -533.303,Z 1018.992,A 0.000,B 0.000,C 90.000,E1 34.532} C_DIS
LIN {X -0.213,Y -528.413,Z 1018.987,A 0.000,B 0.000,C 90.000,E1 33.706} C_DIS
LIN {X 0.011,Y -524.097,Z 1018.983,A 0.000,B 0.000,C 90.000,E1 32.959} C_DIS
LIN {X 0.026,Y -518.610,Z 1018.978,A 0.000,B 0.000,C 90.000,E1 32.084} C_DIS
LIN {X -0.109,Y -514.682,Z 1018.975,A 0.000,B 0.000,C 90.000,E1 31.514} C_DIS
LIN {X -0.104,Y -510.418,Z 1018.972,A 0.000,B 0.000,C 90.000,E1 30.924} C_DIS
LIN {X -0.127,Y -505.915,Z 1018.969,A 0.000,B 0.000,C 90.000,E1 30.335} C_DIS
LIN {X -0.181,Y -501.082,Z 1018.965,A 0.000,B 0.000,C 90.000,E1 29.745} C_DIS
LIN {X -0.091,Y -494.487,Z 1018.961,A 0.000,B 0.000,C 90.000,E1 28.999} C_DIS
LIN {X -0.007,Y -489.179,Z 1018.958,A 0.000,B 0.000,C 90.000,E1 28.409} C_DIS
LIN {X -0.162,Y -482.053,Z 1018.954,A 0.000,B 0.000,C 90.000,E1 27.719} C_DIS
LIN {X -0.056,Y -472.083,Z 1018.949,A 0.000,B 0.000,C 90.000,E1 26.744} C_DIS
LIN {X -0.029,Y -464.609,Z 1018.945,A 0.000,B 0.000,C 90.000,E1 26.052} C_DIS
LIN {X -0.203,Y -458.530,Z 1018.942,A 0.000,B 0.000,C 90.000,E1 25.540} C_DIS
LIN {X 0.109,Y -449.434,Z 1018.937,A 0.000,B 0.000,C 90.000,E1 24.719} C_DIS
LIN {X -0.066,Y -428.386,Z 1018.927,A 0.000,B 0.000,C 90.000,E1 22.898} C_DIS
LIN {X 0.214,Y -415.293,Z 1018.920,A 0.000,B 0.000,C 90.000,E1 21.589} C_DIS
LIN {X -0.064,Y -402.570,Z 1018.912,A 0.000,B 0.000,C 90.000,E1 20.248} C_DIS
LIN {X -0.090,Y -398.480,Z 1018.910,A 0.000,B 0.000,C 90.000,E1 19.758} C_DIS
LIN {X 0.112,Y -393.828,Z 1018.906,A 0.000,B 0.000,C 90.000,E1 19.033} C_DIS
LIN {X 0.094,Y -392.345,Z 1018.904,A 0.000,B 0.000,C 90.000,E1 18.725} C_DIS
LIN {X -0.119,Y -391.630,Z 1018.903,A 0.000,B 0.000,C 90.000,E1 18.489} C_DIS
LIN {X -0.094,Y -391.260,Z 1018.902,A 0.000,B 0.000,C 90.000,E1 18.308} C_DIS
LIN {X -0.144,Y -391.025,Z 1018.900,A 0.000,B 0.000,C 90.000,E1 17.946} C_DIS
LIN {X -0.098,Y -390.931,Z 1018.898,A 0.000,B 0.000,C 90.000,E1 17.583} C_DIS
LIN {X 0.085,Y -391.572,Z 1018.892,A 0.000,B 0.000,C 90.000,E1 16.496} C_DIS
LIN {X 0.056,Y -396.756,Z 1018.866,A 0.000,B 0.000,C 90.000,E1 11.895} C_DIS
LIN {X -0.068,Y -404.162,Z 1018.841,A 0.000,B 0.000,C 90.000,E1 7.352} C_DIS
LIN {X -0.153,Y -411.405,Z 1018.822,A 0.000,B 0.000,C 90.000,E1 3.898} C_DIS
LIN {X -0.147,Y -414.551,Z 1018.814,A 0.000,B 0.000,C 90.000,E1 2.522} C_DIS
LIN {X -0.130,Y -416.754,Z 1018.810,A 0.000,B 0.000,C 90.000,E1 1.835} C_DIS
LIN {X -0.103,Y -418.563,Z 1018.808,A 0.000,B 0.000,C 90.000,E1 1.489} C_DIS
LIN {X -0.080,Y -420.804,Z 1018.806,A 0.000,B 0.000,C 90.000,E1 1.146} C_DIS
LIN {X 0.155,Y -422.876,Z 1018.805,A 0.000,B 0.000,C 90.000,E1 0.859} C_DIS
LIN {X -0.072,Y -426.755,Z 1018.803,A 0.000,B 0.000,C 90.000,E1 0.573} C_DIS
LIN {X -0.165,Y -428.548,Z 1018.802,A 0.000,B 0.000,C 90.000,E1 0.458} C_DIS
LIN {X 0.082,Y -437.723,Z 1018.799,A 0.000,B 0.000,C 90.000,E1 359.885} C_DIS
LIN {X 0.090,Y -449.191,Z 1018.796,A 0.000,B 0.000,C 90.000,E1 359.198} C_DIS
LIN {X -0.165,Y -464.236,Z 1018.791,A 0.000,B 0.000,C 90.000,E1 358.339} C_DIS
LIN {X -0.185,Y -480.809,Z 1018.785,A 0.000,B 0.000,C 90.000,E1 357.364} C_DIS
LIN {X 0.120,Y -489.017,Z 1018.783,A 0.000,B 0.000,C 90.000,E1 356.846} C_DIS
LIN {X 0.074,Y -498.581,Z 1018.779,A 0.000,B 0.000,C 90.000,E1 356.274} C_DIS
LIN {X -0.106,Y -509.698,Z 1018.775,A 0.000,B 0.000,C 90.000,E1 355.584} C_DIS
LIN {X -0.232,Y -518.834,Z 1018.772,A 0.000,B 0.000,C 90.000,E1 354.951} C_DIS
LIN {X -0.120,Y -524.814,Z 1018.769,A 0.000,B 0.000,C 90.000,E1 354.489} C_DIS
LIN {X 0.193,Y -533.446,Z 1018.765,A 0.000,B 0.000,C 90.000,E1 353.742} C_DIS
LIN {X 0.225,Y -540.399,Z 1018.762,A 0.000,B 0.000,C 90.000,E1 353.109} C_DIS
LIN {X 0.090,Y -546.880,Z 1018.758,A 0.000,B 0.000,C 90.000,E1 352.470} C_DIS
LIN {X 0.068,Y -552.999,Z 1018.754,A 0.000,B 0.000,C 90.000,E1 351.781} C_DIS
LIN {X -0.073,Y -556.490,Z 1018.752,A 0.000,B 0.000,C 90.000,E1 351.376} C_DIS
END
